# B&R Automation Studio project TD52 (part 109)

#### DefaultGTCyclic.st - Cyclic code
```iecst
(*******************************************************************************
DefaultGT		value set

This code is confidential and proprietary to the INNIO Company.
It may not be used in any form, or reproduced in any manner,
without the express written permission of the INNIO Company.
Copyright, INNIO Company, 2025

Customized modifications: -
------------------------

History:
-------
V3.99.0		18.09.2012	Denk	new
V04.03.00	02.07.2015	Denk 	Backfire device for 4 gaslines and prechamber
V04.04.00	02.12.2016	Denk 	IN_GT.tSIFA_BOV.Di added
V04.07.00   04.04.2019	Zengerer ParaFactoryDefaults in Init, against missing values at upgrade engines
V04.07.01   06.06.2019	Zengerer ParaFactoryDefaults in Init
V04.25.00	17.12.2025	Theobald With SafetyPLC the gas safety device signals will not be set

Instructions for use:
--------------------
- Default TRUE setting for not existing Di's

Outstandings:
------------

*******************************************************************************)

PROGRAM _CYCLIC

	(* Default TRUE setting for not existing Di's *)
	IN_GT.tDiffPrct_TC2.Di			:= IN_GT.tDiffPrct_TC2.Di 			OR NOT IN_GT.tDiffPrct_TC2.GoodQual;
	IN_GT.tGndFailure_TC2.Di		:= IN_GT.tGndFailure_TC2.Di 		OR NOT IN_GT.tGndFailure_TC2.GoodQual;
	IN_GT.tGT1_SafeDevOK.Di			:=(IN_GT.tGT1_SafeDevOK.Di 			OR NOT IN_GT.tGT1_SafeDevOK.GoodQual) AND NOT IN_GT.bSafetyPLC_Active; 	(* SAFETY PLC *)
	IN_GT.tGT2_SafeDevOK.Di			:=(IN_GT.tGT2_SafeDevOK.Di 			OR NOT IN_GT.tGT2_SafeDevOK.GoodQual) AND NOT IN_GT.bSafetyPLC_Active;	(* SAFETY PLC *)
	IN_GT.tFlairRdy.Di				:= IN_GT.tFlairRdy.Di 				OR NOT IN_GT.tFlairRdy.GoodQual;
	IN_GT.tRelGasPlant.Di			:= IN_GT.tRelGasPlant.Di 			OR NOT IN_GT.tRelGasPlant.GoodQual;
	IN_GT.tPr_GT_MinBefCompr.Di		:= IN_GT.tPr_GT_MinBefCompr.Di 		OR NOT IN_GT.tPr_GT_MinBefCompr.GoodQual;
	IN_GT.tT_GT_Ok.Di				:= IN_GT.tT_GT_Ok.Di 				OR NOT IN_GT.tT_GT_Ok.GoodQual;
	IN_GT.tGT_GC_Fail.Di			:= IN_GT.tGT_GC_Fail.Di 			OR NOT IN_GT.tGT_GC_Fail.GoodQual;
	IN_GT.tGT_FlairFail.Di			:= IN_GT.tGT_FlairFail.Di 			OR NOT IN_GT.tGT_FlairFail.GoodQual;
	IN_GT.tGT_FlareOpMod.Di			:= IN_GT.tGT_FlareOpMod.Di 			OR NOT IN_GT.tGT_FlareOpMod.GoodQual;
	IN_GT.tPr_PCG_Min.Di			:= IN_GT.tPr_PCG_Min.Di 			OR NOT IN_GT.tPr_PCG_Min.GoodQual;
	IN_GT.tOlShortCirc_TC2.Di		:= IN_GT.tOlShortCirc_TC2.Di 		OR NOT IN_GT.tOlShortCirc_TC2.GoodQual;
	IN_GT.tGenPrctTrip_TC2.Di		:= IN_GT.tGenPrctTrip_TC2.Di 		OR NOT IN_GT.tGenPrctTrip_TC2.GoodQual;
	IN_GT.tPr_GT1_Min.Di			:= IN_GT.tPr_GT1_Min.Di 			OR NOT IN_GT.tPr_GT1_Min.GoodQual;
	IN_GT.tPr_GT2_Min.Di			:= IN_GT.tPr_GT2_Min.Di 			OR NOT IN_GT.tPr_GT2_Min.GoodQual;
	IN_GT.tPr_GT1_Max.Di			:= IN_GT.tPr_GT1_Max.Di 			OR NOT IN_GT.tPr_GT1_Max.GoodQual;
	IN_GT.tPr_GT2_Max.Di			:= IN_GT.tPr_GT2_Max.Di 			OR NOT IN_GT.tPr_GT2_Max.GoodQual;
	IN_GT.tSafetyLoop_Eng.Di		:= IN_GT.tSafetyLoop_Eng.Di 		OR NOT IN_GT.tSafetyLoop_Eng.GoodQual;
	IN_GT.tP_GT_Max_Backfire.Di		:= IN_GT.tP_GT_Max_Backfire.Di 		OR NOT IN_GT.tP_GT_Max_Backfire.GoodQual;
	IN_GT.tPCG_GC_Fail.Di			:= IN_GT.tPCG_GC_Fail.Di 			OR NOT IN_GT.tPCG_GC_Fail.GoodQual;
	IN_GT.tPCG_GC_Oil_Min.Di		:= IN_GT.tPCG_GC_Oil_Min.Di 		OR NOT IN_GT.tPCG_GC_Oil_Min.GoodQual;
	IN_GT.tGT_BackFireDev.Di		:= IN_GT.tGT_BackFireDev.Di 		OR NOT IN_GT.tGT_BackFireDev.GoodQual;
	IN_GT.tGT1_1_BackFireDev.Di		:= IN_GT.tGT1_1_BackFireDev.Di 		OR NOT IN_GT.tGT1_1_BackFireDev.GoodQual;
	IN_GT.tGT1_2_BackFireDev.Di		:= IN_GT.tGT1_2_BackFireDev.Di 		OR NOT IN_GT.tGT1_2_BackFireDev.GoodQual;
	IN_GT.tGT1_3_BackFireDev.Di		:= IN_GT.tGT1_3_BackFireDev.Di 		OR NOT IN_GT.tGT1_3_BackFireDev.GoodQual;
	IN_GT.tGT1_4_BackFireDev.Di		:= IN_GT.tGT1_4_BackFireDev.Di 		OR NOT IN_GT.tGT1_4_BackFireDev.GoodQual;
	IN_GT.tPCbComp_BackFireDev.Di 	:= IN_GT.tPCbComp_BackFireDev.Di 	OR NOT IN_GT.tPCbComp_BackFireDev.GoodQual;
	IN_GT.tPCaComp_BackFireDev.Di	:= IN_GT.tPCaComp_BackFireDev.Di 	OR NOT IN_GT.tPCaComp_BackFireDev.GoodQual;
	IN_GT.tRelMainGVext.Di			:= IN_GT.tRelMainGVext.Di 			OR NOT IN_GT.tRelMainGVext.GoodQual;
	IN_GT.tPr_PCGBefComp_Lo.Di		:= IN_GT.tPr_PCGBefComp_Lo.Di 		OR NOT IN_GT.tPr_PCGBefComp_Lo.GoodQual;
	IN_GT.tT_PCGAfComp_Hi.Di		:= IN_GT.tT_PCGAfComp_Hi.Di 		OR NOT IN_GT.tT_PCGAfComp_Hi.GoodQual;
	IN_GT.tGT_AirSupply_LoLo.Di		:= IN_GT.tGT_AirSupply_LoLo.Di		OR NOT IN_GT.tGT_AirSupply_LoLo.GoodQual;
	IN_GT.tPr_GT1_1_Max.Di			:= IN_GT.tPr_GT1_1_Max.Di 			OR NOT IN_GT.tPr_GT1_1_Max.GoodQual;
	IN_GT.tPr_GT1_2_Max.Di			:= IN_GT.tPr_GT1_2_Max.Di 			OR NOT IN_GT.tPr_GT1_2_Max.GoodQual;
	IN_GT.tPr_GT1_3_Max.Di			:= IN_GT.tPr_GT1_3_Max.Di 			OR NOT IN_GT.tPr_GT1_3_Max.GoodQual;
	IN_GT.tPr_GT1_4_Max.Di			:= IN_GT.tPr_GT1_4_Max.Di 			OR NOT IN_GT.tPr_GT1_4_Max.GoodQual;
	IN_GT.tPr_GT1_1_Min.Di			:= IN_GT.tPr_GT1_1_Min.Di 			OR NOT IN_GT.tPr_GT1_1_Min.GoodQual;
	IN_GT.tPr_GT1_2_Min.Di			:= IN_GT.tPr_GT1_2_Min.Di 			OR NOT IN_GT.tPr_GT1_2_Min.GoodQual;
	IN_GT.tPr_GT1_3_Min.Di			:= IN_GT.tPr_GT1_3_Min.Di 			OR NOT IN_GT.tPr_GT1_3_Min.GoodQual;
	IN_GT.tPr_GT1_4_Min.Di			:= IN_GT.tPr_GT1_4_Min.Di 			OR NOT IN_GT.tPr_GT1_4_Min.GoodQual;
	IN_GT.tSIFA_BOV.Di              := IN_GT.tSIFA_BOV.Di       		OR NOT IN_GT.tSIFA_BOV.GoodQual;

END_PROGRAM
```

#### DefaultGTInit.st - Initialization code
```iecst
(********************************************************************
 * COPYRIGHT -- INNIO Company
 ********************************************************************
 * Program: DefaultGT
 * File: DefaultGTInit.st
 * Author: 105046866
 * Created: September 18, 2012
 ********************************************************************
 * Implementation of program DefaultGT
 ********************************************************************)

PROGRAM _INIT

	(* Internal setting *)
	bTestEnabled := FALSE;

	(* V4.07 Para defaults against missing values at upgrade engines *)
	ParaFactoryDefault.iGasTrain_Type 			:= 1;
	ParaFactoryDefault.iGasTrain_Upstream_Type	:= 0;
	ParaFactoryDefault.rGasImp_Prescaling		:= 1;

END_PROGRAM
```

### Program Logical/Gastrain/gasum (IEC) - Gasumschaltung

#### gasumCyclic.st
```iecst
(***************************************************************************
gasum			GASUMSCHALTUNG/GASMISCHBETRIEB MIT KLAPPEN/VENTILEN BZW. TECJET

This code is confidential AND proprietary to the INNIO Company.
It may NOT be used in any form, OR reproduced in any manner,
without the express written permission of the INNIO Company.
Copyright, INNIO Company, 2019

Customized modifications: -
------------------------

History:
-------
V0.1	03.07.98/Pa		erstellt
        24.11.98/Pa		korrekturlesung
V170	06.04.02/LH		überarbeitet
V180	21.01.03/LH		Fehler bei Umschaltung im Stillstand ausgebessert
V183	18.09.03/LH		Kontaktplan --> strukturierten Text
 		02.10.03/LH		Gasmischbetrieb
V2071	22.11.04/LH		Schliessen der entsprechenden Gasstrecke bei Erreichen einer Endlage
                   		Blockierung Mischgasstart
		07.02.05/LH		Gasstrecke nicht mehr anwählbar wenn gestört
		03.03.05/LH		neue Variable "GASUM" eingeführt
V2071b	28.06.05/LH		Task überarbeitet
V210	18.10.04/LH		neu: Mischgasverhältnis manuell einstellbar
V220	28.03.07/LH		Task überarbeitet
V2201	08.08.07/LH		Leistung absenken vor Öffnen der 2. Gasstrecke bei TecJet
V230	16.01.08/LH		Hinweis für Leistungsabsenkung
V2311a	13.05.08/LH		Leistungsabsenkung aus Mischgas wenn Gasmischverhältnis aus Endlage geht
V2.50.0	25.03.2009 		Lettenb.	ssPowerSetpointLimit2 was ssPowerSetpointLimit1 (gasmix->res.2)
V2.50.1 08.07.2009 		Lett./LH Fehler bei Schritt30, bCrossOver und P_FUG ausgebessert
V2.60.0	06.10.2009 		Lettenb	task activation added
V2.60.1	20.01.2010 		lettenb.	INIT: M_GASV1 preset TRUE was FALSE, init vars reduced
V3.20.0	30.09.2010 		Maier(BuR)	M_GSEIN replaced with GCB_ON
V3.99	21-09-2013		Denk 	       	generated for modular software
V3.99.1	14-03-2013		Denk 	       	rFeedbFlap1,rFeedbFlap2,rGT_RatioMix_Set changed from Para to IN-structure
V4.00.00 25-02-2014		Denk/Zengerer  	new interface IN_GT.bGT_SelectRatioMix for DI 'MISCH', FA_M_GASV1, V2 parameter limitation
V4.03.00 29-05-2015		Denk	       	Bugfix, FA_M_GASV2.Hy soll immer 0 sein. Wie bei XT3.
		 02-07-2015		Denk 			Bugfix, 3321 NOT activ when gastrain 2 is active. NOT was missing --> NOT MM2VIS.bMsg1028
		 								Warnings FOR 4 gaslines bMsg2694-2696 added
V4.04.00 06.02.2017		Denk			Bugfix, IN_GT.bIdx_Leanox_Act deleted, changed to IN_GT.bLeanox_Active
V4.05.00 12-10-2017		Zengerer  		Prepare vor standard with tCustAnaIn[1] or IN_GT.rGT_RatioMix_Set, to select the customized setpoint value for ssRatioMix  [0-1]
V4.11.00 17-03-2022		Zuschnig	Use standard label from customized modul for gasmixing setpoint
		 18-03-2022		Zuschnig	Removed fixed spare parameter and customized analog input
V4.13.00 20-06-2023		Zuschnig  	Added standardized AI input for gas mixing ratio
		 20-12-2023		Zuschnig	Prevent division by zero

Instructions for use:
--------------------
activate task if used with Parameter

Outstandings:
------------

****************************************************************************)

(* Übersicht Gasumschaltung *)

(*
           +---------------------------------+                              Umschaltung mit Klappen/Ventilen
           !                                 !                              ohne Rückmeld. und guter Gasqualität
           V                                 V
    +-------------+   +-------------+   +-------------+   +-------------+   Umschaltung mit Klappen/Ventilen
    ! GAS1_2|GAS1 !<->!    GAS2     !<->!    GAS4     !<->!    GAS3     !   ohne Rückmeldung und
    +-------------+   +-------------+   +-------------+   +-------------+   schlechter Gasqualität
           A                                                      A
           !          +-------------------------------+           !         Umschaltung bzw. Gasmischbetrieb mit
           +--------->!           GAS1_3              !<----------+         Klappen/Ventilen mit Rückmeldung
                      +-------------------------------+                     oder mit TecJet

****************************************************************************)
PROGRAM _CYCLIC

(*task activation *)
IF NOT Para.bGT_MixActive THEN
	RETURN;
END_IF

	IF	NOT Para.bTJ_Exist	THEN
		T_GAS1;										(* Klappen-Umschaltzeit [sec], Parameter Eingabe in sec *)
		T_GAS2;										(* Klappen-Umschaltzeit [sec], Parameter Eingabe in sec *)
		T_GAS3;										(* Klappen-Umschaltzeit [sec], Parameter Eingabe in sec *)
		T_GAS4;										(* Klappen-Umschaltzeit [sec], Parameter Eingabe in sec *)
		T_GAS1_4;									(* Klappen-Umschaltzeit [sec], Parameter Eingabe in sec *)
		T_GAS4_1;									(* Klappen-Umschaltzeit [sec], Parameter Eingabe in sec *)
		T_IMPULS;									(* Stellimpuls Klappen  [sec], Parameter Eingabe in sec *)
		T_PAUSE;									(* Pausenzeit Klappen   [sec], Parameter Eingabe in sec *)

		FA_GAS1_2.In		:=	X_GMISCH_2;			(* Gas quality [0-1 = 0-100%] *)
		FA_GAS1_2.Gw		:=	0;					(* GW hohe Qual. [0-1 = 0-100%], Parameter Eingabe in 0-100% *)
		FA_GAS1_2.Hy		:=	0;					(* HY hohe Qual. [0-1 = 0-100%], Parameter Eingabe in 0-100% *)
		FA_GAS1_2;
		GAS1_2_HQ			:=	FA_GAS1_2.Q;		(* GAS1_2 mit hoher Qualität *)

		mit_RM				:=	FALSE;				(* Rückmeldung von Klappen/Ventilen vorhanden *)
		RM_KL1				:=	0;					(* RM Klappe/Ventil Gasstrecke 1 *)
		RM_KL2				:=	0;					(* RM Klappe/Ventil Gasstrecke 2 *)

	END_IF;
	(* bis hier eventuell löschen ------------------------------------------------------------------------------------------------------- *)

	(* Gas mixing setpoint from MM Customized, or directliy connected here with Customized AI[x]  *)
	IF  IN_GT.bOptGT_RatioMix_Set THEN
		X_SOLLW			:=	REAL_TO_INT(LIMIT(0.0, IN_GT.rGT_RatioMix_Set, 1.0) * 1000);	(* Ratio mix from customized module -> 0 - 1 = 0 - 100% *)
	ELSE
		X_SOLLW			:=	REAL_TO_INT(LIMIT(0.0, IN_GT.tGT_RatioMix_Set.Ai, 1.0) * 1000); (* Ratio mix from AI standard label -> 0 - 1 = 0 - 100% *)
	END_IF

	MISCH				:=  IN_GT.tGT_SelectRatioMix.Di;									(* Digital input to select gas mixing (1-3 or 1_2-3) *)
	GUMSCH 				:= 	IN_GT.tGT_TypSwitch.Di;											(* Digital input to select gas type switching *)

	FA_M_GASV1.In		:=	REAL_TO_INT(OUT_GT.rGT_RatioMix * 1000);						(* MAX-Grenzwert Mischrate *)
	FA_M_GASV1.Gw		:=	1000;															(* GW Mischrate [0-1000 = 100%], Parameter Eingabe in 0-100% *)
	FA_M_GASV1.Hy		:=	5;																(* HY Mischrate [0-1000 = 100%], Parameter Eingabe in 0-100% *)
	FA_M_GASV1;																				(* --> Schliessen Gasventil 1 *)

	FA_M_GASV2.In		:=	REAL_TO_INT(OUT_GT.rGT_RatioMix * 1000);						(* MIN-Grenzwert Mischrate *)
	FA_M_GASV2.Gw		:=	0;																(* GW Mischrate [0-1000 = 100%], Parameter Eingabe in 0-100% *)
	FA_M_GASV2.Hy		:=	5;																(* HY Mischrate [0-1000 = 100%], Parameter Eingabe in 0-100% *)
	FA_M_GASV2;																				(* --> Schliessen Gasventil 2 *)

	(* Copy of input variables to local *)			//!!! new
	ssRatioMix 			:= REAL_TO_INT(OUT_GT.rGT_RatioMix * 1000);
	M_BTRB 				:= IN_GT.tEng_Run.Do;
	GCB_ON 				:= IN_GT.tGCB_On.Di;
	M_GASV 				:= OUT_GT.bGV_On;
	AUTGAS				:= OUT_GT.bSelGasTypAut;
	GAS1_2_MAN			:= OUT_GT.bSelGasTyp0;
	GAS1_3_MAN			:= OUT_GT.bSelGasTypMix;
	GAS1				:= OUT_GT.bSelGasTyp1;
	GAS2				:= OUT_GT.bSelGasTyp2;
	GAS3				:= OUT_GT.bSelGasTyp3;
	GAS4				:= OUT_GT.bSelGasTyp4;
	bLeanoxActive		:= IN_GT.bLeanox_Active;
	l_einst_a			:= IN_GT.bLeanox_Man;
	M_NANF				:= IN_GT.bEng_Dem_EPS;
	M_GDMI1W			:= MM2VIS.bMsg3221;
	M_GDMI1_1W			:= MM2VIS.bMsg2694;
	M_GDMI1_2W			:= MM2VIS.bMsg2695;
	M_GDMI1_3W			:= MM2VIS.bMsg2696;
	M_GDMI2W			:= MM2VIS.bMsg3222;
	anz_gasart			:= INT_TO_USINT(Para.iIdx_Gastyp);
	bTecJetOn			:= Para.bTJ_Exist;
	GASV1				:= OUT_GT.tGV1_Open.Do;
	GASV2				:= OUT_GT.tGV2_Open.Do;
	p_ist				:= REAL_TO_INT(IN_GT.rP_Act_Norm_Filt * IN_GT.rP_Nom);
	bSetMix_Man			:= bGT_RatioMix_Man_Set;						// From Visu
	bMisch1_2_Man		:= bGT_QualMix_Man_Set;							// From Visu
	ssSetMix_Man		:= REAL_TO_INT((rGT_RatioMix_Man_Set) * 1000);	// From Visu
	KL1_AUF				:= IN_GT.tGT_Flap1_Opened.Di;					//will be no IN in future
	KL1_ZU				:= IN_GT.tGT_Flap1_Closed.Di;					//will be no IN in future
	KL2_AUF				:= IN_GT.tGT_Flap2_Opened.Di;					//will be no IN in future
	KL2_ZU				:= IN_GT.tGT_Flap2_Closed.Di;					//will be no IN in future
	GAS1_2				:= OUT_GT.bGT_Ipol12Active;

	//There will be NO spare power reduction in future. One standard for gasmixing
	//--> required setpoint will be setted via OUT_GT.rP_Red_GasSwitch in %
	sel_PowerSetpointLimit := 1;												    				(*Auswahl Reserve-Red: 1 = P-Red Reserve 1
																										 					2 = P-Red Reserve 2
																															3 = P-Red Reserve 3 *)
	ssPowerSetpointLimit:=  4000; 																	(* Text: P_401 !     *)(* Reduktionsleistung für Öffnen 2. Gasstr.[kW] *)
																									(* P_40 Text2! *)

//	TOF_FUGITIV.PT 		:= 	INT_TO_UDINT(LIMIT(5, SPS_REZP1, 5))*100;								//existing code
	TOF_FUGITIV.PT 		:= 	500;	    															(* Verweilzeit auf Reduktionleistung [sec], Parameter Eingabe in sec *)
	TON_P_FUG.PT		:=	200;																	(* Beruhigungzeit bei Erreichen von Pred [0,01sec] *)

	T_TJ				:=	10;																		(* Änderungsgeschwindigkeit Mischrate [promill/sec] *)

	GU_TJ				:=	bTecJetOn;																(* Gasumschaltung mit TecJet *)
	GASUM				:=	TRUE;																	(* Freigabe Gasumschaltung *)
	GAS1_3				:=	GU_TJ OR mit_RM;														(* Freigabe Gasmischung *)
	bGasMixture			:=	GU_TJ AND GASUM;														(* Freigabe Mischgas für VISU (Vers. > 2.10 --> "engine data") *)

						(* Auswahl Treibgasart *)

	FG_MIX				:=	M_BTRB AND (GCB_ON OR FG_MIX);						(* Freigabe Mischgasbetrieb *)

	IF	NOT FG_MIX	THEN
						MISCH				:=	0;
						IF	M_GASV	THEN										(* Gasart fixieren! *)
											GUMSCH				:=	GUMSCH_OLD;
						ELSE				GUMSCH_OLD			:=	GUMSCH;
						END_IF;
	END_IF;

	MISCHGAS			:=	(AUTGAS AND     MISCH OR GAS1_3_MAN)AND(GAS1_3 OR   bLeanoxActive) AND NOT l_einst_a AND NOT M_NANF AND FG_MIX ;

	GASSTR_1			:=	(AUTGAS AND NOT MISCH AND NOT GUMSCH OR(GAS1       AND NOT GAS1_2)
	                                                             OR(GAS1_2_MAN AND     GAS1_2))AND NOT l_einst_a AND NOT M_NANF;
	GASSTR_2			:=	(AUTGAS AND NOT MISCH AND     GUMSCH OR GAS3                      )AND NOT l_einst_a      OR M_NANF;

	IF	(M_GDMI1W OR M_GDMI1_1W OR M_GDMI1_2W OR M_GDMI1_3W) AND ANW_GST2	THEN	(* Gasstrecke 1 nicht anwählbar! *)
						MISCHGAS			:=	0;
						GASSTR_1			:=	0;
						GASSTR_2			:=	1;
	END_IF;

	IF	M_GDMI2W AND NOT UW_GST2 OR NOT(anz_gasart > 2)	THEN						(* Gasstrecke 2 nicht anwählbar! *)
						MISCHGAS			:=	0;
						GASSTR_1			:=	1;
						GASSTR_2			:=	0;
	END_IF;

						(* Schrittkette *)

	CASE	step OF	00:	(* Initialisierung (GUI_0) *)
						IF	 ssRatioMix = 0 AND bTecJetOn OR KL1_AUF AND KL2_AUF	THEN
											step				:=	10;			(* 10 = GAS1 / 20 = GAS3 *)
	(* bis hier bearbeiten -------------------------------------------------------------------------------------------------------------- *)
											IF	bTecJetOn	THEN
																step				:=	10;
											END_IF;
											GUI_7				:=	1;			(* Initialisierung abgeschlossen ! *)
						END_IF;

					10:	(* Treibgas 1 (GU2_7) *)
						IF	 (GASSTR_2 OR MISCHGAS) AND GAS1_3	THEN
											step				:=	11;
						ELSIF GASSTR_2 AND NOT GAS1_3	THEN
											step				:=	12;
						END_IF;
						IF	  GASSTR_2 AND M_NANF AND NOT GCB_ON AND KL2_AUF AND NOT GU_TJ	THEN
											step				:=	20;
						END_IF;

					11:	(* Treibgas 1 --> Mischgas (GU13_0) *)
						IF	(KL2_ZU AND NOT GU_TJ) OR NOT M_GASV OR P_FUG	THEN
											step				:=	30;
						END_IF;

					12:	(* Schliessen Klappe 2 (GU1_0) *)
						IF	KL2_ZU OR NOT M_GASV	THEN
											step				:=	13;
						END_IF;

					13:	(* Gasart 1 (GU1_1) *)
						IF	(T_GAS1_OK AND NOT GAS1_2_HQ) OR NOT M_GASV	THEN
											step				:=	14;
						END_IF;
						IF	(T_GAS1_4_OK AND GAS1_2_HQ) OR KL2_AUF	THEN
											step				:=	15;
						END_IF;

					14:	(* Gasart 2 (GU1_2) *)
						IF	KL2_AUF OR (T_GAS1_4_OK AND GAS1_2_HQ)	THEN
											step				:=	15;
						ELSIF NOT T_GAS1_4_OK AND GAS1_2_HQ	THEN
											step				:=	13;
						END_IF;

					15:	(* Gasart 4 (GU1_3) *)
						IF	T_GAS4_OK OR NOT M_GASV	THEN
											step				:=	16;
						ELSIF NOT KL2_AUF AND NOT GAS1_2_HQ	THEN
											step				:=	14;
						END_IF;

					16:	(* Gasart 3 (GU1_4) *)
						IF	KL1_ZU OR NOT M_GASV	THEN
											step				:=	20;
						END_IF;

					17:	(* Öffnen Klappe 2 (GU31_0) *)
						IF	KL2_AUF OR GU_TJ	THEN
											step				:=	18;
						END_IF;

					18:	(* Schliessen Klappe 1 (GU31_1) *)
						IF	KL1_ZU OR NOT M_GASV OR GU_TJ	THEN
											step				:=	19;
						END_IF;

					19:	(* Mischgas --> Treibgas 2 (GU31_2) *)
						IF	ssRatioMix = 1000 OR NOT GU_TJ	THEN
											step				:=	20;
						ELSIF	MISCHGAS OR GASSTR_1	THEN
											step				:=	30;
						END_IF;

					20:	(* Treibgas 2 (GU1_7) *)
						IF	 (MISCHGAS OR GASSTR_1) AND GAS1_3	THEN
											step				:=	21;
						ELSIF GASSTR_1 AND NOT GAS1_3	THEN
											step				:=	22;
						END_IF;

					21:	(* Treibgas 2 --> Mischgas (GU23_0) *)
						IF	KL1_ZU AND NOT GU_TJ OR NOT M_GASV OR P_FUG	THEN
											step				:=	30;
						END_IF;

					22:	(* Schliessen Klappe 1 (GU2_0) *)
						IF	KL1_ZU OR NOT M_GASV	THEN
											step				:=	23;
						END_IF;

					23:	(* Gasart 3 (GU2_1) *)
						IF	T_GAS3_OK OR NOT M_GASV OR KL1_AUF	THEN
											step				:=	24;
						END_IF;

					24:	(* Gasart 4 (GU2_2) *)
						IF	KL1_AUF	THEN
											IF	NOT GAS1_2_HQ	THEN
																step				:=	25;
											ELSIF	T_GAS4_1_OK OR NOT M_GASV	THEN
																step				:=	26;
											END_IF;
						END_IF;

					25:	(* Gasart 2 (GU2_3) *)
						IF	T_GAS2_OK OR (T_GAS4_1_OK AND GAS1_2_HQ) OR NOT M_GASV	THEN
											step				:=	26;
						ELSIF NOT T_GAS4_1_OK AND GAS1_2_HQ	THEN
											step				:=	24;
						END_IF;

					26:	(* Gasart 1 (GU2_4) *)
						IF	KL2_ZU OR NOT M_GASV	THEN
											step				:=	10;
						ELSIF NOT T_GAS2_OK AND NOT GAS1_2_HQ	THEN
											step				:=	25;
						END_IF;

					27:	(* Öffnen Klappe 1 (GU32_0) *)
						IF	KL1_AUF OR GU_TJ	THEN
											step				:=	28;
						END_IF;

					28:	(* Schliessen Klappe 2 (GU32_1) *)
						IF	KL2_ZU OR NOT M_GASV OR GU_TJ	THEN
											step				:=	29;
						END_IF;

					29:	(* Mischgas --> Treibgas 1 (GU32_2) *)
						IF	ssRatioMix = 0 OR NOT GU_TJ	THEN
											step				:=	10;
						ELSIF	GASSTR_2 OR MISCHGAS	THEN
											step				:=	30;
						END_IF;

					30:	(* Mischgas (GU3_7) *)
						IF		GASSTR_2	THEN
											step				:=	17;
						ELSIF	GASSTR_1	THEN
											step				:=	27;
						END_IF;
						IF	(X_SOLLW > (FA_M_GASV2.Gw + FA_M_GASV2.Hy)) AND NOT GASV2 AND M_GASV AND NOT P_FUG AND GU_TJ	THEN
											step				:=	11;
						END_IF;
						IF	(X_SOLLW < (FA_M_GASV1.Gw - FA_M_GASV1.Hy)) AND NOT GASV1 AND M_GASV AND NOT P_FUG AND GU_TJ	THEN
											step				:=	21;
						END_IF;

	END_CASE;

						(* Schrittkettenmerker *)

	zw					:= 1;
	FOR	i				:= 1 TO step	BY 1 DO
						zw				:=	zw * 2;
	END_FOR;
	FA_CONV_1.Word		:= UDINT_TO_UINT(zw);
	FA_CONV_1;

	zw					:= 1;
	FOR i				:= 17 TO step	BY 1 DO
						zw				:=	zw * 2;
	END_FOR;
	IF	step < 16 THEN	zw				:=	0;
	END_IF;
	FA_CONV_2.Word		:= UDINT_TO_UINT(zw);
	FA_CONV_2;

	GUI_0				:= FA_CONV_1.Bit00;										(* Initialisierung *)
	GUI_1				:= FA_CONV_1.Bit01;										(* Initialisierung *)
	GUI_2				:= FA_CONV_1.Bit02;										(* Initialisierung *)
	GUI_3				:= FA_CONV_1.Bit03;										(* Initialisierung *)
	GUI_4				:= FA_CONV_1.Bit04;										(* Initialisierung *)
	GUI_5				:= FA_CONV_1.Bit05;										(* Initialisierung *)
	GUI_6				:= FA_CONV_1.Bit06;										(* Initialisierung *)
	muell				:= FA_CONV_1.Bit07;
	muell				:= FA_CONV_1.Bit08;
	muell				:= FA_CONV_1.Bit09;
	GU2_7				:= FA_CONV_1.Bit10;										(* Treibgas 1 *)
	GU13_0				:= FA_CONV_1.Bit11;										(* Treibgas 1 --> Mischgas *)
	GU1_0				:= FA_CONV_1.Bit12;										(* Schliessen Klappe/Ventil 2 *)
	GU1_1				:= FA_CONV_1.Bit13;										(* Gasart 1 / Gasart 1_2 *)
	GU1_2				:= FA_CONV_1.Bit14;										(* Gasart 2 *)
	GU1_3				:= FA_CONV_1.Bit15;										(* Gasart 4 *)
	GU1_4				:= FA_CONV_2.Bit00;										(* Gasart 3 *)
	GU31_0				:= FA_CONV_2.Bit01;										(* Öffnenen Klappe/Ventil 2 *)
	GU31_1				:= FA_CONV_2.Bit02;										(* Schliessen Klappe/Ventil 1 *)
	GU31_2				:= FA_CONV_2.Bit03;										(* Mischgas --> Treibgas 2 *)
	GU1_7				:= FA_CONV_2.Bit04;										(* Treibgas 2 *)
	GU23_0				:= FA_CONV_2.Bit05;										(* Treibgas 2 --> Mischgas *)
	GU2_0				:= FA_CONV_2.Bit06;										(* Schliessen Klappe/Ventil 2 *)
	GU2_1				:= FA_CONV_2.Bit07;										(* Gasart 3 *)
	GU2_2				:= FA_CONV_2.Bit08;										(* Gasart 4 *)
	GU2_3				:= FA_CONV_2.Bit09;										(* Gasart 2 *)
	GU2_4				:= FA_CONV_2.Bit10;										(* Gasart 1 / Gasart 1_2 *)
	GU32_0				:= FA_CONV_2.Bit11;										(* Öffnenen Klappe/Ventil 1 *)
	GU32_1				:= FA_CONV_2.Bit12;										(* Schliessen Klappe/Ventil 2 *)
	GU32_2				:= FA_CONV_2.Bit13;										(* Mischgas --> Treibgas 1 *)
	GU3_7				:= FA_CONV_2.Bit14;										(* Mischgas *)
	muell				:= FA_CONV_2.Bit15;

						(* Setzen der Steuerbefehle *)

	FG_GST				:=	GUI_7 AND(GU2_7 OR GU1_7 OR M_BTRB OR GU3_7 AND GAS1_3);(* Freigabe Gasstrecke (pb6!) *)

	FG_MISCH			:=	GU3_7;												(* Freigabe Gasmischregler (reg_in!)*)

	V_GVD				:=	GU23_0;												(* Vorhalte Gasverdichter *)

	ANW_GST2			:=	GU1_7 OR GU23_0 OR GU2_0;							(* Anwahl Gasstrecke 2 *)
	UW_GST2				:=	NOT(GU2_7 OR GU13_0 OR GU1_0);						(* Überwachung Gasstrecke 2 *)

	M_GASV1				:=	NOT ANW_GST2 AND(									(* Anwahl Gasventil 1 *)
							GU_TJ OR NOT KL1_ZU)AND(NOT
							GU_TJ OR NOT FA_M_GASV1.Q);
	M_GASV2				:=	UW_GST2 AND(										(* Anwahl Gasventil 2 *)
							GU_TJ OR NOT KL2_ZU)AND(NOT
							GU_TJ OR NOT FA_M_GASV2.Q);

	bCrossOver			:=	GASV1 AND GASV2 AND bTecJetOn;						(* Gasmischung aktiv für TecJet's *)

	M_AWGAS1			:=	(GU1_1 OR GU2_4 OR NOT M_GASV2)AND NOT GAS1_2;		(* Anwahl Gas1 *)
	M_AWGAS1_2			:=	(GU1_1 OR GU2_4 OR NOT M_GASV2)AND     GAS1_2;		(* Anwahl Interpolation *)
	M_AWGAS1_3			:=	(GU3_7 OR GU31_2 OR GU32_2)AND bCrossOver OR(		(* Anwahl Mischgas *)
							GU31_0 OR GU31_1 OR
							GU32_0 OR GU32_1)AND NOT bTecJetOn;

	M_AWGAS1			:=	M_AWGAS1 OR M_AWGAS1_2 OR M_AWGAS1_3;				(* Anwahl Gas1 *)
	M_AWGAS2			:=	(GU1_2 OR GU2_3);									(* Anwahl Gas2 *)
	M_AWGAS3			:=	(GU1_4 OR GU2_1 OR NOT M_GASV1);					(* Anwahl Gas3 *)
	M_AWGAS4			:=	(GU1_3 OR GU2_2);									(* Anwahl Gas4 *)

	IF	M_GASV AND (GU13_0 OR GU23_0) AND NOT bCrossOver AND bTecJetOn	THEN(* Entlasten für Öffnen anderen Gasstrecke *)
						FUGITIV				:=	1;								(* Anforderung Leistungsreduktion *)
	ELSE				FUGITIV				:=	0;
	END_IF;

	TOF_FUGITIV.IN := FUGITIV;
	TOF_FUGITIV.PT := MAX(TOF_FUGITIV.PT, ((MAX((1000 - (FA_M_GASV1.Gw - FA_M_GASV1.Hy)), ((FA_M_GASV2.Gw + FA_M_GASV2.Hy) - 0))/MAX(1, T_TJ))*100));
	TOF_FUGITIV();
	sel_PowerSetpointLimit := LIMIT(0, sel_PowerSetpointLimit, 3);
	bPowerSetpointLimit    :=((p_ist > ssPowerSetpointLimit) OR bPowerSetpointLimit) AND TOF_FUGITIV.Q AND (sel_PowerSetpointLimit > 0);

	TON_P_FUG.IN := ((p_ist <= ssPowerSetpointLimit) OR TON_P_FUG.IN) AND
					((p_ist - ssPowerSetpointLimit) < ssPowerSetpointLimit/50);
	TON_P_FUG();

	IF	TON_P_FUG.Q AND FUGITIV	THEN
						P_FUG				:=	1;								(* Reduktionsleistung erreicht *)
	ELSE				P_FUG				:=	0;
	END_IF;

	IF		GASSTR_1 OR GU32_2 OR GUI_0	THEN									(* Gasmischverhältnis für GAS1 *)
						X_SOLLW				:=	0;
	ELSIF	GASSTR_2 OR GU31_2	THEN											(* Gasmischverhältnis für GAS3 *)
						X_SOLLW				:=	1000;
	ELSE				X_SOLLW				:=	MUX(BOOL_TO_SINT(bSetMix_Man),	(* Gasmischverhältnis für Mischbetrieb *)
												X_SOLLW, ssSetMix_Man);
	END_IF;

	IF	M_GASV AND (l_einst_a OR GU13_0 OR GU23_0)	THEN						(* Gasmischverhältnis fixieren! *)
						X_SOLLW				:=	X_SOLLW_OLD;
	ELSE				X_SOLLW_OLD			:=	X_SOLLW;
	END_IF;

	IF	NOT M_GASV OR (GU31_2 AND M_NANF AND NOT GCB_ON)	THEN				(* disable ramp fub *)
						RAMPE_X_SOLLW.enable := FALSE;
	ELSE				RAMPE_X_SOLLW.enable := TRUE;							(* enable ramp fub *)
						RAMPE_X_SOLLW.Rise	 := INT_TO_UINT(					(* pos. change of gas mixture 0,1%/sec *)
												LIMIT(0,T_TJ*BOOL_TO_INT(NOT l_einst_a),10));
						RAMPE_X_SOLLW.Sink	 := INT_TO_UINT(					(* neg. change of gas mixture 0,1%/sec *)
												LIMIT(0,T_TJ*BOOL_TO_INT(NOT l_einst_a),10));
	END_IF;
	RAMPE_X_SOLLW.TC_Time:= 100;												(* FUB is working in 100ms task		*)
	RAMPE_X_SOLLW.In	 := X_SOLLW;
	RAMPE_X_SOLLW();

	OUT_GT.rGT_MixSet	:= 	INT_TO_REAL(LIMIT(0, RAMPE_X_SOLLW.Out, 1000)) / 1000;	(* Sollwert für Gasmischverhältnis *)
//	ssSetMix			:=	LIMIT(0, RAMPE_X_SOLLW.Out, 1000);						(* Sollwert für Gasmischverhältnis *)		//Existing code

						(* Steuerbefehle für Klappen/Ventile *)

	KL1AUF_1			:=	GUI_0 AND NOT GU_TJ;								(* Initialisierung *)
	KL1ZU_1				:=	GUI_0 AND NOT GU_TJ AND NULL;						(* Initialisierung *)
	KL2AUF_1			:=	GUI_0 AND NOT GU_TJ;								(* Initialisierung *)
	KL2ZU_1				:=	GUI_0 AND NOT GU_TJ AND NULL;						(* Initialisierung *)

	KL1AUF_2			:=	(GU2_1 OR GU2_2 AND NOT KL1_AUF)					(* Treibgas 2 --> Treibgas 1 (getaktet) *)
							AND NOT l_einst_a;
	KL1ZU_2				:=	(GU1_3 AND KL2_AUF OR GU1_4)						(* Treibgas 1 --> Treibgas 2 (getaktet) *)
							AND NOT l_einst_a;
	KL2AUF_2			:=	(GU1_1 OR GU1_2 OR GU1_3 AND NOT KL2_AUF)			(* Treibgas 1 --> Treibgas 2 (getaktet) *)
							AND NOT l_einst_a;
	KL2ZU_2				:=	(GU2_2 AND KL1_AUF AND GAS1_2_HQ OR GU2_3 OR GU2_4)	(* Treibgas 2 --> Treibgas 1 (getaktet) *)
							AND NOT l_einst_a;

	KL1AUF_3			:=	GU32_0 AND NOT GU_TJ AND NOT l_einst_a;				(* Mischgas --> Treibgas 1 (getaktet) *)
	KL1ZU_3				:=	GU31_1 AND NOT GU_TJ AND NOT l_einst_a;				(* Mischgas --> Treibgas 2 (getaktet) *)
	KL2AUF_3			:=	GU31_0 AND NOT GU_TJ AND NOT l_einst_a;				(* Mischgas --> Treibgas 2 (getaktet) *)
	KL2ZU_3				:=	GU32_1 AND NOT GU_TJ AND NOT l_einst_a;				(* Mischgas --> Treibgas 1 (getaktet) *)

	KL1AUF_4			:=	KL1AUF_2 AND NOT M_GASV OR							(* Treibgas 2 --> Treibgas 1 (direkt) *)
							GU32_0 AND NOT M_GASV AND NOT GU_TJ;				(* Mischgas --> Treibgas 1 (direkt) *)

	KL1ZU_4				:=	KL1ZU_2 AND NOT M_GASV OR							(* Treibgas 1 --> Treibgas 2 (direkt) *)
							GU31_1 AND NOT M_GASV AND NOT GU_TJ OR				(* Mischgas --> Treibgas 2 (direkt) *)
							GU1_7 AND NOT KL1_ZU AND NOT GU_TJ OR				(* Treibgas 2 (direkt) *)
							GU23_0 AND M_GASV AND NOT GU_TJ OR					(* Treibgas 2 --> Mischgas (direkt) *)
							GU2_0;												(* Treibgas 2 --> Treibgas 1 (direkt) *)

	KL2AUF_4			:=	KL2AUF_2 AND NOT M_GASV OR							(* Treibgas 1 --> Treibgas 2 (direkt) *)
							GU31_0 AND NOT M_GASV AND NOT GU_TJ OR				(* Mischgas --> Treibgas 2 (direkt) *)
							GU2_7 AND NOT KL2_AUF AND NOT GU_TJ;				(* Treibgas 1 (direkt) *)

	KL2ZU_4				:=	GU13_0 AND M_GASV AND NOT GU_TJ OR					(* Treibgas 1 --> Mischgas (direkt) *)
							GU1_0;												(* Treibgas 1 --> Treibgas 2 (direkt) *)

	KL1AUF_5			:=	GU3_7 AND NOT l_einst_a;							(* Gasmischbetrieb (Schrittregler!) *)
	KL1ZU_5				:=	GU3_7 AND NOT l_einst_a AND KL2_AUF;				(* Gasmischbetrieb (Schrittregler!) *)
	KL2AUF_5			:=	GU3_7 AND NOT l_einst_a;							(* Gasmischbetrieb (Schrittregler!) *)
	KL2ZU_5				:=	GU3_7 AND NOT l_einst_a AND KL1_AUF;				(* Gasmischbetrieb (Schrittregler!) *)

	IF	GU2_7 OR GU1_7 OR (KL1_AUF AND KL2_AUF)	THEN
						count				:=	0;
	END_IF;
	IF		(GU1_1 OR GU1_2)	THEN
						IF	count > (MIN(T_GAS1, T_GAS1_4) * 10)	THEN		(* Zeit Gasart 1 *)
											T_GAS1_OK			:=	1;
						END_IF;
						IF	count > (MAX(T_GAS1_4, T_GAS1) * 10)	THEN		(* Zeit Gasart 1 mit hoher Qualität *)
											T_GAS1_4_OK			:=	1;
						END_IF;
						count				:=	count + BOOL_TO_INT(KL2AUF_2);
	END_IF;
	IF	GU1_3 AND KL2_AUF 	THEN
						IF	count > (T_GAS4 * 10)	THEN						(* Zeit Gasart 4 (Treibgas 1 --> Treibgas 2) *)
											T_GAS4_OK			:=	1;
						END_IF;
						count				:=	count + BOOL_TO_INT(KL1ZU_2);
	END_IF;
	IF	GU2_1	THEN
						IF	count > (T_GAS3 * 10)	THEN						(* Zeit Gasart 3 *)
											T_GAS3_OK			:=	1;
						END_IF;
						count				:=	count + BOOL_TO_INT(KL1AUF_2);
	END_IF;
	IF	GU2_2 AND KL1_AUF OR GU2_3 OR GU2_4	THEN
						IF	count > (MIN(T_GAS4_1, T_GAS2) * 10)	THEN		(* Zeit Gasart 4 (Treibgas 2 --> Treibgas 1) *)
											T_GAS4_1_OK			:=	1;
						END_IF;
						IF	count > (MAX(T_GAS2, T_GAS4_1) * 10)	THEN		(* Zeit Gasart 2 *)
											T_GAS2_OK			:=	1;
						END_IF;
						count				:=	count + BOOL_TO_INT(KL2ZU_2);
	END_IF;
	IF	GU2_7 OR GU1_7	THEN
						T_GAS1_OK			:=	0;
						T_GAS1_4_OK			:=	0;
						T_GAS4_OK			:=	0;
						T_GAS3_OK			:=	0;
						T_GAS4_1_OK			:=	0;
						T_GAS2_OK			:=	0;
	END_IF;

						(* Taktgenerierung für Stellbefehle *)

	IMPULS				:=	T_IMPULS * 10;
	PAUSE				:=	T_PAUSE * 10;
	IF	count_st > (IMPULS + PAUSE)	THEN
						count_st			:=	0;
	END_IF;
	IF	count_st > 0	THEN
						STELL				:=	1;
	END_IF;
	IF	count_st > IMPULS	THEN
						STELL				:=	0;
	END_IF;
	count_st			:=	count_st + 1;

						(* Stellbefehle Klappen/Ventile *)

	KL1AUF				:=	(((KL1AUF_2 OR KL1AUF_3) AND STELL) OR (KL1AUF_5 AND GAS2_MIN) OR KL1AUF_4 OR KL1AUF_1) AND NOT KL1_AUF;
	KL1ZU				:=	(((KL1ZU_2  OR KL1ZU_3)  AND STELL) OR (KL1ZU_5  AND GAS2_PLU) OR KL1ZU_4  OR KL1ZU_1)  AND NOT KL1_ZU;
	KL2AUF				:=	(((KL2AUF_2 OR KL2AUF_3) AND STELL) OR (KL2AUF_5 AND GAS2_PLU) OR KL2AUF_4 OR KL2AUF_1) AND NOT KL2_AUF;
	KL2ZU				:=	(((KL2ZU_2  OR KL2ZU_3)  AND STELL) OR (KL2ZU_5  AND GAS2_MIN) OR KL2ZU_4  OR KL2ZU_1)  AND NOT KL2_ZU;

						(* Ventilstellwerte (mA-Vorgabe) *)

	IF	KL1AUF	THEN	count1				:=	count1 + 1;
	END_IF;
	IF	KL1ZU	THEN	count1				:=	count1 - 1;
	END_IF;
	IF	KL2AUF	THEN	count2				:=	count2 + 1;
	END_IF;
	IF	KL2ZU	THEN	count2				:=	count2 - 1;
	END_IF;
	count1				:=	LIMIT(0, count1, 1000);
	count2				:=	LIMIT(0, count2, 1000);
	SW_KL1				:=	count1;
	SW_KL2				:=	count2;

						(* Rückmeldungen Ventilendstellungen *)

	IF	NOT mit_RM	THEN
						RM_KL1				:=	SW_KL1;
						RM_KL2				:=	SW_KL2;
						IF	RM_KL1 < 1		THEN
											KL1_ZU				:=	1;
						ELSE				KL1_ZU				:=	0;
						END_IF;
						IF	RM_KL1 > 999	THEN
											KL1_AUF				:=	1;
						ELSE				KL1_AUF				:=	0;
						END_IF;
						IF	RM_KL2 < 1		THEN
											KL2_ZU				:=	1;
						ELSE				KL2_ZU				:=	0;
						END_IF;
						IF	RM_KL2 > 999	THEN
											KL2_AUF				:=	1;
						ELSE				KL2_AUF				:=	0;
						END_IF;
	END_IF;

						(* Gasverbräuche (gmv_ber) *)

	GAS1_VB	:=	BOOL_TO_INT(GASV1) * (
							BOOL_TO_INT(NOT GU_TJ)*(RM_KL1 + 1000-RM_KL2*BOOL_TO_INT(GASV2)) +
							BOOL_TO_INT(GU_TJ)*(1000 - ssRatioMix));
	GAS2_VB	:=	BOOL_TO_INT(GASV2) * (
							BOOL_TO_INT(NOT GU_TJ)*(RM_KL2 + 1000-RM_KL1*BOOL_TO_INT(GASV1)) +
							BOOL_TO_INT(GU_TJ)*ssRatioMix);

	(* Leistungsreduktionen *)
	(* Power reduction gas switching for opening second gastrain *)
	IF (ssPowerSetpointLimit <= 0.0) OR (IN_GT.rP_Act_Norm_Filt = 0.0) OR (IN_GT.rP_Nom = 0.0) THEN			//new
		OUT_GT.rP_Red_GasSwitch := 0.0;
	ELSE
		OUT_GT.rP_Red_GasSwitch := 1 - LIMIT(0.0, (Para.rP_GT_SetLim / (IN_GT.rP_Act_Norm_Filt * IN_GT.rP_Nom)), 0.5);
	END_IF;

(* Copy local output variables to global *)
	bGT_MixingEna 				:= bGasMixture;				(* Visu *)
	OUT_GT.bGT2_Select 			:= ANW_GST2;
	OUT_GT.bGT_Rel 				:= FG_GST;
	OUT_GT.bGT_RelMixing		:= FG_MISCH;
	OUT_GT.bGasMixingActive		:= bCrossOver;
	OUT_GT.bGT_SelGas1			:= M_AWGAS1;
	OUT_GT.bGT_SelGas2			:= M_AWGAS2;
	OUT_GT.bGT_SelGas3			:= M_AWGAS3;
	OUT_GT.bGT_SelGas4			:= M_AWGAS4;
    OUT_GT.tGT_Flap1_Open.Do 	:= KL1AUF;			//will be no Out in future
	OUT_GT.tGT_Flap1_Close.Do	:= KL1ZU;			//will be no Out in future
	OUT_GT.tGT_Flap2_Open.Do	:= KL2AUF;			//will be no Out in future
	OUT_GT.tGT_Flap2_Close.Do	:= KL2ZU;			//will be no Out in future
	OUT_GT.bGT_TypSwhActive		:= GASUM;

END_PROGRAM
```

#### gasumInit.st
```iecst
PROGRAM _INIT

END_PROGRAM
```

#### gasum.var
```iecst
VAR
	anz_gasart : USINT; (* number of gas types *)
	AUTGAS : BOOL := 0; (* AUTOMATIK Gasumschaltung *)
	bLeanoxActive : BOOL; (* TRUE=leanox controller is active *)
	bMisch1_2_Man : BOOL; (* 1=gas quality manual *)
	bPowerSetpointLimit : BOOL;
	bTecJetOn : BOOL; (* TRUE=gas inject valves are active *)
	count : INT := 0;
	count_st : INT := 0;
	count1 : INT := 0; (* Klappensimulation *)
	count2 : INT := 0; (* Klappensimulation *)
	FA_CONV_1 : WDtoBIT;
	FA_CONV_2 : WDtoBIT;
	FA_GAS1_2 : GR_MAXR;
	FA_M_GASV1 : GR_MAX;
	FA_M_GASV2 : GR_MIN;
	FG_GST : BOOL := 0; (* Freigabe Gasstrecke *)
	FG_MISCH : BOOL := 0; (* Freigabe Gasmischregler *)
	FUGITIV : BOOL := 0; (* Anforderung Leistungsreduktion *)
	GAS1 : BOOL := 0; (* Gasart 1 *)
	GAS1_2 : BOOL; (*param.interpolation gas1 & 2 active from CH4(or CV)*)
	GAS1_2_MAN : BOOL := 0; (* Gasart 0 manuell *)
	GAS1_3_MAN : BOOL := 0; (* Mischgas manuell *)
	GAS2 : BOOL := 0; (* Gasart 2 *)
	GAS2_MIN : BOOL := 0; (* weniger Treibgas 2 *)
	GAS2_PLU : BOOL := 0; (* mehr Treibgas 2 *)
	GAS3 : BOOL := 0; (* Gasart 3 *)
	GAS4 : BOOL := 0; (* Gasart 4 *)
	GASSTR_1 : BOOL := 0; (* Anwahl Gasstrecke 1 *)
	GASSTR_2 : BOOL := 0; (* Anwahl Gasstrecke 2 *)
	GASV1 : BOOL := 0; (* Gasventil 1 *)
	GASV2 : BOOL := 0; (* Gasventil 2 *)
	GCB_ON : BOOL := FALSE; (*Generatorschalter EIN (TK#3 synchron)*)
	GU1_0 : BOOL := 0; (* Schrittkettenmerker *)
	GU1_1 : BOOL := 0; (* Schrittkettenmerker *)
	GU1_2 : BOOL := 0; (* Schrittkettenmerker *)
	GU1_3 : BOOL := 0; (* Schrittkettenmerker *)
	GU1_4 : BOOL := 0; (* Schrittkettenmerker *)
	GU1_7 : BOOL := 0; (* Schrittkettenmerker *)
	GU2_0 : BOOL := 0; (* Schrittkettenmerker *)
	GU2_1 : BOOL := 0; (* Schrittkettenmerker *)
	GU2_2 : BOOL := 0; (* Schrittkettenmerker *)
	GU2_3 : BOOL := 0; (* Schrittkettenmerker *)
	GU2_4 : BOOL := 0; (* Schrittkettenmerker *)
	GU2_7 : BOOL := 0; (* Schrittkettenmerker *)
	GU3_7 : BOOL := 0; (* Schrittkettenmerker *)
	GU13_0 : BOOL := 0; (* Schrittkettenmerker *)
	GU23_0 : BOOL := 0; (* Schrittkettenmerker *)
	GU31_0 : BOOL := 0; (* Schrittkettenmerker *)
	GU31_1 : BOOL := 0; (* Schrittkettenmerker *)
	GU31_2 : BOOL := 0; (* Schrittkettenmerker *)
	GU32_0 : BOOL := 0; (* Schrittkettenmerker *)
	GU32_1 : BOOL := 0; (* Schrittkettenmerker *)
	GU32_2 : BOOL := 0; (* Schrittkettenmerker *)
	GUI_0 : BOOL := 0; (* Schrittkettenmerker *)
	GUI_1 : BOOL := 0; (* Schrittkettenmerker *)
	GUI_2 : BOOL := 0; (* Schrittkettenmerker *)
	GUI_3 : BOOL := 0; (* Schrittkettenmerker *)
	GUI_4 : BOOL := 0; (* Schrittkettenmerker *)
	GUI_5 : BOOL := 0; (* Schrittkettenmerker *)
	GUI_6 : BOOL := 0; (* Schrittkettenmerker *)
	GUI_7 : BOOL := 0; (* Gasumschaltung INIT abgeschlossen *)
	GUMSCH : BOOL := 0; (* Gasumschaltung auf 2.tes Treibgas *)
	GUMSCH_OLD : BOOL;
	i : INT;
	IMPULS : INT; (* Stellimpuls *)
	KL1_AUF : BOOL := 0; (* RM Gasklappe 1 offen *)
	KL1_ZU : BOOL := 0; (* RM Gasklappe 1 geschlossen *)
	KL1AUF : BOOL := 0; (* GASKLAPPE 1 AUFFAHREN *)
	KL1AUF_1 : BOOL := 0; (* Klappensteuerbefehl *)
	KL1AUF_2 : BOOL := 0; (* Klappensteuerbefehl *)
	KL1AUF_3 : BOOL := 0; (* Klappensteuerbefehl *)
	KL1AUF_4 : BOOL := 0; (* Klappensteuerbefehl *)
	KL1AUF_5 : BOOL := 0; (* Klappensteuerbefehl *)
	KL1ZU : BOOL := 0; (* GASKLAPPE 1 ZUFAHREN *)
	KL1ZU_1 : BOOL := 0; (* Klappensteuerbefehl *)
	KL1ZU_2 : BOOL := 0; (* Klappensteuerbefehl *)
	KL1ZU_3 : BOOL := 0; (* Klappensteuerbefehl *)
	KL1ZU_4 : BOOL := 0; (* Klappensteuerbefehl *)
	KL1ZU_5 : BOOL := 0; (* Klappensteuerbefehl *)
	KL2_AUF : BOOL := 0; (* RM Gasklappe 2 offen *)
	KL2_ZU : BOOL := 0; (* RM Gasklappe 2 geschlossen *)
	KL2AUF : BOOL := 0; (* GASKLAPPE 2 AUFFAHREN *)
	KL2AUF_1 : BOOL := 0; (* Klappensteuerbefehl *)
	KL2AUF_2 : BOOL := 0; (* Klappensteuerbefehl *)
	KL2AUF_3 : BOOL := 0; (* Klappensteuerbefehl *)
	KL2AUF_4 : BOOL := 0; (* Klappensteuerbefehl *)
	KL2AUF_5 : BOOL := 0; (* Klappensteuerbefehl *)
	KL2ZU : BOOL := 0; (* GASKLAPPE 2 ZUFAHREN *)
	KL2ZU_1 : BOOL := 0; (* Klappensteuerbefehl *)
	KL2ZU_2 : BOOL := 0; (* Klappensteuerbefehl *)
	KL2ZU_3 : BOOL := 0; (* Klappensteuerbefehl *)
	KL2ZU_4 : BOOL := 0; (* Klappensteuerbefehl *)
	KL2ZU_5 : BOOL := 0; (* Klappensteuerbefehl *)
	l_einst_a : BOOL; (* TRUE=leanox controller in manual *)
	M_BTRB : BOOL := 0; (* Aggregat in BETRIEB *)
	M_GASV : BOOL := 0; (* Gasventile EIN *)
	M_GDMI1W : BOOL := 0; (*3221 Gasdruck 1 minimum *)
	M_GDMI1_1W : BOOL := 0; (*2694 Gasdruck 1 Linie 1 minimum *)
	M_GDMI1_2W : BOOL := 0; (*2695 Gasdruck 1 Linie 2 minimum *)
	M_GDMI1_3W : BOOL := 0; (*2696 Gasdruck 1 Linie 3 minimum *)
	M_GDMI2W : BOOL := 0; (*3222 Gasdruck 2 minimum *)
	M_NANF : BOOL := 0; (* Notstromanforderung *)
	MISCH : BOOL := 0; (* Mischgas *)
	MISCHGAS : BOOL := 0; (* Anwahl Mischgas *)
	mit_RM : BOOL := 0; (* mit RM Klappe/Ventil *)
	muell : BOOL := 0; (* GARBAGE BIT *)
END_VAR
VAR CONSTANT
	NULL : BOOL := 0; (* immer NULL *)
END_VAR
VAR
	P_FUG : BOOL := 0; (* Reduktionsleistung erreicht *)
	p_ist : INT; (* actual filtered power [kW] T= 1sec *)
	PAUSE : INT; (* Pausenzeit *)
	RAMPE_X_SOLLW : RAMPE;
	RM_KL1 : INT; (* RM Klappe/Ventil 1 *)
	RM_KL2 : INT; (* RM Klappe/Ventil 2 *)
	sel_PowerSetpointLimit : INT;
	ssPowerSetpointLimit : INT;
	ssRatioMix : INT; (* gas mixture rate after ramp fub *)
	ssSetMix_Man : INT;
	STELL : BOOL := 0; (* Stellimpuls *)
	step : INT := 0; (* Schrittvariable *)
	SW_KL1 : INT := 0; (* Sollwert Ventil 1 *)
	SW_KL2 : INT := 0; (* Sollwert Ventil 2 *)
	T_GAS1 : INT; (* Zeitwert *)
	T_GAS1_4 : INT; (* Zeitwert *)
	T_GAS1_4_OK : BOOL := FALSE;
	T_GAS1_OK : BOOL := FALSE;
	T_GAS2 : INT; (* Zeitwert *)
	T_GAS2_OK : BOOL := FALSE;
	T_GAS3 : INT; (* Zeitwert *)
	T_GAS3_OK : BOOL := FALSE;
	T_GAS4 : INT; (* Zeitwert *)
	T_GAS4_1 : INT; (* Zeitwert *)
	T_GAS4_1_OK : BOOL := FALSE;
	T_GAS4_OK : BOOL := FALSE;
	T_IMPULS : INT; (* Zeitwert *)
	T_PAUSE : INT; (* Zeitwert *)
	T_TJ : INT := 10; (* Rampenzeit Tecjet *)
	TOF_FUGITIV : TOF_10ms;
	TON_P_FUG : TON_10ms;
	X_SOLLW : INT; (* SOLLWERT Mischgasverhältnis *)
	X_SOLLW_OLD : INT;
	zw : UDINT;
END_VAR
```

### Program Logical/Gastrain/gas_rail (IEC) - gas rail control

#### gas_railCyclic.st
```iecst
(*******************************************************************************
gas_rail

This code is confidential and proprietary to the INNIO Company.
It may not be used in any form, or reproduced in any manner,
without the express written permission of the INNIO Company.
Copyright, INNIO Company, 2019

Customized modifications: -
------------------------

History:
-------
V04.03.00	20.01.2015  Denk 		Porting J920 for XT4
			07.04.2016  Denk		Change logic for A2240 ("...ja, lass es uns so machen, dass es eine Freigabebedingung gibt. 2240 soll nur auslösen, wenn es keine Messsignalstörung 2567 gibt..." E-mail 07.04.2016 Klaus Spyra)
V04.04.00	04.07.2016	Denk		Change logic for bAMM_T_GR_HiHi. Additional: AND OUT_GT.tGV1_Open.Do;
V04.05.00	20.03.2017	Denk		SWAT920: Several changes regarding new specification
V04.05.01	24.10.2017	Zingerle	Reduction with difference pressure minimum, implemented
V04.05.02	01.03.2018	Denk		Reduction with difference pressure minimum, Spec. change and validation changes
V04.05.03	23.03.2018	Denk		Perm2 change because of new Perm_GT2 file
V04.07.00	04.07.2018	Denk		Bugfix, Anzeige Leistungsreduktion Gasdruck min.
V04.10.00	05.08.2020	Zuschnig	Included 50ms filtered for boost pressure for differential pressure limit monitoring
V04.11.00	20.01.2022	Zuschnig	Update gas rail pressure power reduction

Instructions for use:
--------------------
*******************************************************************************)
PROGRAM _CYCLIC

	(*--------------------------------------------------------------*)
	(* RESET of alarms and warnings 								*)
	(*--------------------------------------------------------------*)
	bAMM_Pr_GR_I_MS			:= FALSE;
	bAMM_Pr_GR_II_MS		:= FALSE;
	bAMM_Pr_GR_I_LoLo		:= FALSE;
	bAMM_Pr_GR_I_HiHi		:= FALSE;
	bAMM_DPr_GR_I_LoLo		:= FALSE;
	bAMM_DPr_GR_I_HiHi		:= FALSE;
	bAMM_DPr_GR_I_Lo		:= FALSE;
	bAMM_DPr_GR_I_Hi		:= FALSE;
	bAMM_T_GR_MS			:= FALSE;
	bAMM_T_GR_LoLo			:= FALSE;
	bAMM_T_GR_HiHi			:= FALSE;
	bAMM_T_GR_Lo			:= FALSE;
	bAMM_T_GR_Hi			:= FALSE;
	bAMM_Pr_MGT_a_Filt_Min	:= FALSE;

	rP_norm_red_1				:= 1.0;
	rP_norm_red_2				:= 1.0;
	OUT_GT.rP_Red_Pr_GR_Norm	:= 1.0;

	(************************************************************************************************************************************)
	(************************              				  error monitoring		 	             	           **************************)
	(************************************************************************************************************************************)
	IF IN_GT.tPB2MM.bParaSetupOk THEN

		(*----------------------------------------------------------*)
		(* measurement signal failure 								*)
		(*----------------------------------------------------------*)
		bAMM_Pr_GR_I_MS		:= Para.bPr_GR_I_Exist 	AND NOT IN_GT.tPr_GR_I.GoodQual;		(* W2443 *)
		bAMM_Pr_GR_II_MS	:= Para.bPr_GR_II_Exist	AND NOT IN_GT.tPr_GR_II.GoodQual;		(* W2444 *)
		bAMM_Pr_GR_I_II_MS  := bAMM_Pr_GR_I_MS 		AND 	bAMM_Pr_GR_II_MS; 				(* A2309 *)
		bAMM_T_GR_MS		:= Para.bT_GR_Exist 	AND NOT IN_GT.tT_GR.GoodQual;			(* W2567 *)

		(* Release monitoring	*)
		xTOF_AMM_Pr_GR_I_MS(IN 	:= bAMM_Pr_GR_I_MS,	 PT:= T#10s);	(* TOF because of filtered signals *)
		xTOF_AMM_Pr_GR_II_MS(IN	:= bAMM_Pr_GR_II_MS, PT:= T#10s);
		xTOF_AMM_T_GR_MS(IN  	:= bAMM_T_GR_MS, 	 PT:= T#10s);

		bRelMon_Pr_GR_I		:= Para.bPr_GR_I_Exist 	AND NOT xTOF_AMM_Pr_GR_I_MS.Q;
		bRelMon_Pr_GR_II	:= Para.bPr_GR_II_Exist AND NOT xTOF_AMM_Pr_GR_II_MS.Q;
		bRelMon_Pr_GR_Avg	:= bRelMon_Pr_GR_I 		OR 		bRelMon_Pr_GR_II;
		bRelMon_T_GR		:= Para.bT_GR_Exist 	AND NOT xTOF_AMM_T_GR_MS.Q;

		(*----------------------------------------------------------*)
		(* check gas rail pressure sensor deviation					*)
		(*----------------------------------------------------------*)
		LCRMAF_PGR_Deviation.x := ABS(IN_GT.tPr_GR_I.Ai - IN_GT.tPr_GR_II.Ai);

		LCRMAF_PGR_Deviation();

		xGR_MAX_Deviation.In := LCRMAF_PGR_Deviation.y;
		xGR_MAX_Deviation.Gw := 0.130;	(* 130mbar *)
		xGR_MAX_Deviation.Hy := 0.03; 	(* 30mbar *)
		xGR_MAX_Deviation();

		bDevP_GR_TooHigh := xGR_MAX_Deviation.Q AND bRelMon_Pr_GR_I AND bRelMon_Pr_GR_II;

		(*----------------------------------------------------------*)
		(* gas rail pressure limit monitoring						*)
		(*----------------------------------------------------------*)
		xGR_MAX_AGRPR(In := IN_GT.tPr_GR_I.Ai, Gw := Para.rPr_GR_HiHi, Hy := 0.0);

		bAMM_Pr_GR_I_HiHi 	:= xGR_MAX_AGRPR.Q AND bRelMon_Pr_GR_I;		(* A2244 *)

		(*----------------------------------------------------------*)
		(* differential pressure limit monitoring					*)
		(*----------------------------------------------------------*)
		xGR_MAX_APDPR(In := (rPr_GR_Avg - xFILTER_R_P2s_50ms.Out), Gw := Para.rPr_GR_Diff_HiHi, Hy := 0.0);
		xGR_MIN_APDPR(In := (rPr_GR_Avg - xFILTER_R_P2s_50ms.Out), Gw := Para.rPr_GR_Diff_LoLo, Hy := 0.0);

		bAMM_DPr_GR_I_HiHi	:= xGR_MAX_APDPR.Q AND OUT_GT.tGV1_Open.Do;	(* A2248 *)
		bAMM_DPr_GR_I_LoLo	:= xGR_MIN_APDPR.Q AND IN_GT.tGCB_On.Di ;	(* A2249 *)

		(*----------------------------------------------------------*)
		(* gas rail temperature limit monitoring					*)
		(*----------------------------------------------------------*)
		xGR_MAX_WGRTP(In := IN_GT.tT_GR.Ai, Gw := (Para.rT_GR_HiHi - 5.0), Hy := 0.0);
		xGR_MIN_WGRTP(In := IN_GT.tT_GR.Ai, Gw := (Para.rT_GR_LoLo), Hy := 0.0);

		bAMM_T_GR_Hi	:= xGR_MAX_WGRTP.Q AND bRelMon_T_GR AND OUT_GT.tGV1_Open.Do;			(* W2568 *)
		bAMM_T_GR_Lo	:= xGR_MIN_WGRTP.Q AND bRelMon_T_GR AND OUT_GT.tGV1_Open.Do;			(* W2569 *)

		xGR_MAX_AGRTP(In := IN_GT.tT_GR.Ai, Gw := Para.rT_GR_HiHi, Hy := 0.0);

		bAMM_T_GR_HiHi	:= xGR_MAX_AGRTP.Q AND bRelMon_T_GR AND OUT_GT.tGV1_Open.Do;			(* A2240 *)

		(*----------------------------------------------------------*)
		(* gas rail pressure average filtered						*)
		(*----------------------------------------------------------*)
		IF 	  (NOT bRelMon_Pr_GR_I AND NOT bRelMon_Pr_GR_II) THEN	rPr_GR_Avg :=  0;
		ELSIF (NOT bRelMon_Pr_GR_I AND 	   bRelMon_Pr_GR_II) THEN	rPr_GR_Avg :=  IN_GT.tPr_GR_II.Ai;
		ELSIF (	   bRelMon_Pr_GR_I AND NOT bRelMon_Pr_GR_II) THEN	rPr_GR_Avg :=  IN_GT.tPr_GR_I.Ai;
		ELSE
			IF NOT bDevP_GR_TooHigh  THEN
				rPr_GR_Avg := (IN_GT.tPr_GR_I.Ai + IN_GT.tPr_GR_II.Ai ) / 2;
			ELSE
				IF  ABS(IN_GT.tPr_GR_I.Ai - (rPr_MGT_sp + IN_GT.rPr_Baro_Internal)) <  ABS(IN_GT.tPr_GR_II.Ai - (rPr_MGT_sp + IN_GT.rPr_Baro_Internal))  THEN
			 		rPr_GR_Avg := IN_GT.tPr_GR_I.Ai;
				ELSE
					rPr_GR_Avg := IN_GT.tPr_GR_II.Ai;
				END_IF;
			END_IF;
		END_IF;
		OUT_GT.rPr_GR_filt := rPr_GR_Avg;

		(*----------------------------------------------------------*)
		(* gas rail pressure average unfiltered						*)
		(*----------------------------------------------------------*)
		IF 	  (NOT bRelMon_Pr_GR_I AND NOT bRelMon_Pr_GR_II) THEN	rPr_GR_Avg_UF :=  0;
		ELSIF (NOT bRelMon_Pr_GR_I AND 	   bRelMon_Pr_GR_II) THEN	rPr_GR_Avg_UF :=  IN_GT.tPr_GR_II.Unfilt;
		ELSIF (	   bRelMon_Pr_GR_I AND NOT bRelMon_Pr_GR_II) THEN	rPr_GR_Avg_UF :=  IN_GT.tPr_GR_I.Unfilt;
		ELSE
			IF NOT bDevP_GR_TooHigh  THEN
				rPr_GR_Avg_UF := (IN_GT.tPr_GR_I.Unfilt + IN_GT.tPr_GR_II.Unfilt ) / 2;
			ELSE
				IF  ABS(IN_GT.tPr_GR_I.Ai- (rPr_MGT_sp + IN_GT.rPr_Baro_Internal)) <  ABS(IN_GT.tPr_GR_II.Ai - (rPr_MGT_sp + IN_GT.rPr_Baro_Internal))  THEN
			 		rPr_GR_Avg_UF := IN_GT.tPr_GR_I.Unfilt;
				ELSE
					rPr_GR_Avg_UF := IN_GT.tPr_GR_II.Unfilt;
				END_IF;
			END_IF;
		END_IF;
		OUT_GT.rPr_GR_UF := rPr_GR_Avg_UF;

		(*----------------------------------------------------------*)
		(* calculate differential pressure 							*)
		(*----------------------------------------------------------*)
		rPr_MGT_Diff := OUT_GT.rPr_GR_filt - IN_GT.rPr_Ch_P2s_Avg;

		(*------------------------------------------------------------------*)
		(* differential pressure minimum / power reduction					*)
		(*------------------------------------------------------------------*)

		(* charge pressure depending limit calculation *)
		IF bRelMon_Pr_GR_Avg AND OUT_GT.tGV1_Open.Do THEN
			xGR_MIN_Red1_DP(In := (rPr_MGT_Diff / xSigScal_R_DPr_MGT_sp.Y_SCAL), Gw := Perm2.rDPr_limit_pgr_Pred, Hy := rHy_GR_MIN);
			IF xGR_MIN_Red1_DP.Q THEN
				OUT_GT.rP2s_red_1 := (OUT_GT.rPr_GR_filt - (Perm2.rDPr_limit_pgr_Pred * xSigScal_R_DPr_MGT_sp.Y_SCAL));
				rP_norm_red_1	  := LIMIT(0.0, (IN_GT.rP_el_max_red / MAX(1, IN_GT.rP_Nom)), 1.0);
			ELSE
				rP_norm_red_1 := 1.00;
			END_IF;

			IF Para.bPr_GR_red_Exist THEN
				IF ((Para.rPr_GR_red_start - IN_GT.tPr_MGT_a_Filt.Ai) * Para.rP_Pr_GR_red_rate) < 1.0 THEN
					rP_norm_red_2 := LIMIT(0.0, (1 - ((Para.rPr_GR_red_start - IN_GT.tPr_MGT_a_Filt.Ai) * Para.rP_Pr_GR_red_rate)), 1.0);
				ELSE
					rP_norm_red_2 := 1.00;
				END_IF;
			ELSE
				rP_norm_red_2 := 1.00;
			END_IF;

			IF IN_GT.tGCB_On.Di THEN
				OUT_GT.rP_Red_Pr_GR_Norm :=	MIN(rP_norm_red_1, rP_norm_red_2);
			ELSE
				OUT_GT.rP_Red_Pr_GR_Norm	:= 1.0;
			END_IF;

			IF ((IN_GT.tPr_MGT_a_Filt.Ai - (rPr_GR_Avg - IN_GT.rPr_Baro_Internal)) < rPr_GR_Threshold) THEN
				xTP_Pr_MGT_a_Filt_Min(IN := TRUE, PT := T#2s);
			ELSE
				xTP_Pr_MGT_a_Filt_Min(IN := FALSE, PT := T#2s);
			END_IF;

			bAMM_Pr_MGT_a_Filt_Min := xTP_Pr_MGT_a_Filt_Min.Q;
		ELSE
			xTP_Pr_MGT_a_Filt_Min(IN := FALSE, PT := T#2s);
		END_IF;

	END_IF;

END_PROGRAM
```

#### gas_railInit.st
```iecst
(*******************************************************************************
gas_rail		gas rail  					(INIT)

This code is confidential AND proprietary to the INNIO Company.
It may NOT be used in any form, or reproduced in any manner,
without the express written permission of the INNIO Company.
Copyright, INNIO Company, 2019

Customized modifications: -
------------------------

History:
-------
V04.03.00.00  20.01.2015  Denk 		Porting J920 FOR XT4
V04.12.00.00  23.08.2022  Zuschnig	Initialize standard value for power redcution gas rail pressure

Instructions FOR use:
--------------------
*******************************************************************************)
PROGRAM _INIT

	(* check gas pressure sensor deviation *)
	LCRMAF_PGR_Deviation.enable	:= TRUE;	(* *)
	LCRMAF_PGR_Deviation.base	:= 5;		(* *)

	(* Initialize standard value fr power redcution gas rail pressure *)
	IF Perm2.rDPr_limit_pgr_Pred = 0 THEN	Perm2.rDPr_limit_pgr_Pred := 0.7;	END_IF;

END_PROGRAM
```

#### gas_rail.var
```iecst
VAR
	bRelMon_Pr_GR_I : BOOL := FALSE; (*Release monitoring gas sensor 1*)
	bRelMon_Pr_GR_II : BOOL := FALSE; (*Release monitoring gas sensor 2*)
	bRelMon_T_GR : BOOL := FALSE; (*Release monitoring gas rail temperature*)
	LCRMAF_PGR_Deviation : LCRMovAvgFlt;
	xGR_MAX_AGRPR : GR_MAXR := (0); (*FuB*)
	xGR_MAX_AGRTP : GR_MAXR := (0); (*FuB*)
	xGR_MAX_APDPR : GR_MAXR := (0); (*FuB*)
	xGR_MAX_WGRTP : GR_MAXR := (0); (*FuB*)
	xGR_MIN_APDPR : GR_MINR := (0); (*FuB*)
	xGR_MIN_WGRTP : GR_MINR := (0); (*FuB*)
	xTOF_AMM_Pr_GR_II_MS : TOF := (0); (*FuB*)
	xTOF_AMM_Pr_GR_I_MS : TOF := (0); (*FuB*)
	xTOF_AMM_T_GR_MS : TOF := (0); (*FuB*)
	xGR_MAX_Deviation : GR_MAXR;
	rP_norm_red_1 : REAL; (*power reduction boost pressure of the limited power of nominal power  *)
	rP_norm_red_2 : REAL; (*power reduction derating curve for the engine of nominal power  *)
	xGR_MIN_Red1_DP : GR_MINR; (* GR_MIN for power reduction GR *)
	rHy_GR_MIN : REAL := 0.25; (* Gas train diff pressure for power reduction hysteresis *)
	rPr_GR_Threshold : REAL := 0.05; (* Threshold for difference between main gas pressure after filter and gas rail pressure [bar] *)
	xTP_Pr_MGT_a_Filt_Min : TP; (* TP for difference between main gas pressure after filter and gas rail pressure minimum *)
END_VAR
```

### Program Logical/Gastrain/gas_train (IEC) - gas train control

#### gas_trainCyclic.st
```iecst
(*******************************************************************************
gas_train

This code is confidential and proprietary to the INNIO Company.
It may not be used in any form, or reproduced in any manner,
without the express written permission of the INNIO Company.
Copyright, INNIO Company, 2019

Customized modifications: -
------------------------

History:
-------
V3.30.0		06.11.2014  Tinello	NEW specification
V4.03.00  	13.11.2014  Mari 		Porting J920 FOR XT4
			09.02.2014  Denk 		Bugfix, monitoring OF load rejection
			02.06.2015  Denk		MM2VIS.rPr_PCGT_sp, MM2VIS.rPr_MGT_sp now in gas_train task
V4.04.00	03.07.2016	Denk		Blow off valve Open, Spec. change: gasrail pressure > baro pressure + 80mbar (IN_GT.rPr_Baro_Internal + 0.08)
			04.08.2016	Denk		Bugfix, Filterung charge pressure
			15.09.2016	Denk 		set/actual gas pressure comparison, hard coded values changed
			20.10.2016	Tinello		A2271 deleted / A2261 change limit from 60mbar to 100mbar
V4.05.00	24.04.2017	Denk		SWAT 920 Rel.2, A2247 deleted, W2462 new, B2927 new, OUT_GT.bAMM_Pr_MGT_a_Filt_BlockStart new
									SWAT 920 Rel.2, A3377 active > 2MW
			10.07.2017	Denk		SWAT 920 Rel.3, A2257 deleted, W2465 new, B2928 new, OUT_GT.bAMM_Pr_PCGT_a_Filt_BlockStart new
V4.07.00	30.04.2018	Denk		SWAT 920 Rel.5, change A2289 to W2570
									SWAT 920 Rel.5,	deactivation of A3376 when pressure based control is active
									SWAT 920 Rel.5,	W3445 delay time
V4.07.00	10.12.2018	Zengerer 	Gas valve position detection for Requisition standardisation
V4.07.01	28.08.2019	Zengerer 	Upstream Gas valve tGV_Upstream_Open
V4.09.00BETA 02.10./10.07.2019	Ze 	iGasTrain_Upstream_Type.0 corr. basisupdate
		 	21.08.2019	Zengerer 	Alternative path, if NO selection bit from Para.iGasTrain_Upstream_Type is active
		 	19.11.2019	Zengerer 	Customer Main Gas Valve control and position feedback according to updated spec from Lang Thomas
V4.10.00    05.08.2020  Zuschnig    Added control of dome blow off valve
			07.12.2020	Zengerer	IN_GT.tFastStartReq for change according to issue #
V4.11.00	22.06.2021	Arnold		data center serialization: calculation of rPr_MGT_sp based on IN_GT.rPr_Leanox_Set; DBOV different hysteresis and time delay
			20.01.2022	Zuschnig	Update A2289 - Compressed air supply failure
			11.02.2022 	Zuschnig	Remove engine demand for release of upstream gas valve
V4.12.00	22.01.2023	Zuschnig	Add H2 content processing and detection of measurement failure
V4.14.00	06.11.2024	Kafka		fast gastrain for Gen2 type9

Instructions for use:
--------------------
Use UPSTREAM MAIN GAS VALVE OPTION 0 or 1 only (OUT_GT.tGV_Upstream_Open)
UPSTREAM MAIN GAS VALVE OPTION 2  HAS TO BE IMPLEMENTED ACCORDING TO CUSTOMIZED NEEDS in V4.07!
(not global released in V4.07, until sufficient pilot plant installation and testing, according email Hirzinger- Unterrainer, 28.05.2019)

ToDo:
-----

*******************************************************************************)
PROGRAM _CYCLIC

	(*--------------------------------------------------------------*)
	(* RESET of alarms and warnings and pre-settings				*)
	(*--------------------------------------------------------------*)
	bAMM_GT_AirSupply_Lo		:= FALSE;
	bAMM_GT_AirSupply_LoLo		:= FALSE;

	bAMM_DPr_GR_Baro_HiHi		:= FALSE;	(* A2261 *)

	bAMM_Pr_PCGT_Out_MS			:= FALSE;	(* W3448 *)

	bAMM_Pr_MGT_a_Filt_MS		:= FALSE;	(* W2462 *)
	bAMM_Pr_MGT_a_Filt_Lo		:= FALSE;	(* W2535 *)
	bAMM_Pr_MGT_a_Filt_LoLo		:= FALSE;	(* A2243 *)
	bAMM_Pr_MGT_a_Filt_Hi		:= FALSE;	(* W2536 *)
	bAMM_Pr_MGT_a_Filt_HiHi		:= FALSE;	(* A2246 *)
	bAMM_DPr_MGT_SetAct_Hi		:= FALSE;	(* W3444 *)
	bAMM_DPr_MGT_SetAct_HiHi	:= FALSE;	(* A3376 *)

	bAMM_Pr_PCGT_a_Filt_MS		:= FALSE;	(* W2465 *)
	bAMM_Pr_PCGT_a_Filt_Lo		:= FALSE;	(* W2537 *)	(*nicht verwendet*)
	bAMM_Pr_PCGT_a_Filt_LoLo	:= FALSE;	(* A2250 *)	(*nicht verwendet*)
	bAMM_Pr_PCGT_a_Filt_Hi		:= FALSE;	(* W2538 *)
	bAMM_Pr_PCGT_a_Filt_HiHi	:= FALSE;	(* A2251 *)
	bAMM_DPr_PCGT_SetAct_Hi		:= FALSE;	(* W3445 *)
	bAMM_DPr_PCGT_SetAct_HiHi	:= FALSE;	(* A3377 *)

	(* Reset set-/actual-pressure deviation calculation *)
	rDPr_MGT_SetAct				:= 0;
	rDPr_PCGT_SetAct			:= 0;

	(* Mapping of previous parameter for compatibility of visu *)
	Para.bPr_MGT_a_Filt_Exist	:= Para.bPr_GT1_Active;
	Para.rPr_MGT_a_Filt_Hi		:= Para.rPr_GT1_LimHi2;
	Para.rPr_MGT_a_Filt_HiHi	:= Para.rPr_GT1_LimHi1;
	Para.rPr_MGT_a_Filt_Lo		:= Para.rPr_GT1_LimLo2;
	Para.rPr_MGT_a_Filt_LoLo	:= Para.rPr_GT1_LimLo1;

	Para.bPr_PCGT_a_Filt_Exist  := Para.bPr_PCGT_Active;
	Para.rPr_PCGT_a_Filt_Hi		:= Para.rPr_PCGT_LimHi2;
	Para.rPr_PCGT_a_Filt_HiHi	:= Para.rPr_PCGT_LimHi1;
	Para.rPr_PCGT_a_Filt_Lo		:= Para.rPr_PCGT_LimLo2;
	Para.rPr_PCGT_a_Filt_LoLo	:= Para.rPr_PCGT_LimLo1;

	(*--------------------------------------------------------------*)
	(* gas valve			 		 								*)
	(*--------------------------------------------------------------*)
	xTON_GASV_08s(IN:= OUT_GT.tGV1_Open.Do,	PT:= T#8s);
	xTON_GASV_20s(IN:= OUT_GT.tGV1_Open.Do, PT:= T#20s);

	bGASV_Open_8s	:= xTON_GASV_08s.Q;											(* valve opened for  8 seconds *)
	bGASV_Open_20s	:= xTON_GASV_20s.Q;											(* valve opened for 20 seconds *)

	(*--------------------------------------------------------------*)
	(* Filterung charge pressure			 		 								*)
	(*--------------------------------------------------------------*)
	xFILTER_R_P2s_200ms(In := IN_GT.rPr_Ch_P2s_Avg_UF, Filter := 20);
	xFILTER_R_P2s_50ms(In := IN_GT.rPr_Ch_P2s_Avg_UF, Filter := 5);
	xFILTER_R_P2s_500ms(In := IN_GT.rPr_Ch_P2s_Avg_UF, Filter := 50);
	xFILTER_R_P2s_160ms(In := IN_GT.rPr_Ch_P2s_Avg_UF, Filter := 16);

	(*--------------------------------------------------------------*)
	(* Filtering H2 content			 		 								*)
	(*--------------------------------------------------------------*)
	IF Para.bGT_H2Active THEN
		bMSF_H2 := (NOT IN_GT.tGT_H2.GoodQual AND IN_GT.tPB2MM.bParaSetupOk AND NOT IN_GT.bH2_Bus_Active) OR
				   (NOT IN_GT.bH2_Bus_MSF AND IN_GT.tPB2MM.bParaSetupOk AND IN_GT.bH2_Bus_Active);
		(* Measurement signal failure H2 content self-retain *)
		bS_MSF_H2 := bMSF_H2 OR (bS_MSF_H2 AND NOT IN_GT.tAB2GT.bResetWarning);
	ELSE
		bMSF_H2 				:= FALSE;
		bS_MSF_H2				:= FALSE;
	END_IF;

	IF Para.tiFilterConst_H2 = 0 THEN
		xLCRPT1_H2.t := 0.001; (* Filter time constant [s] *)
	ELSE
		xLCRPT1_H2.t := TIME_TO_REAL(Para.tiFilterConst_H2) /1000; (* Filter time constant [s] *)
	END_IF;
	IF NOT Para.bGT_H2Active THEN	(* Switch to zero H2 value in case H2 content measurement is not active *)
		xLCRPT1_H2.x := 0;
	ELSIF bS_MSF_H2 THEN			(* Switch to default H2 value in case of measurement signal failure H2 content *)
		xLCRPT1_H2.x := Para.rGT_H2_DefVal;
	ELSIF NOT IN_GT.bH2_Bus_Active THEN
		xLCRPT1_H2.x := LIMIT(0, IN_GT.tGT_H2.Unfilt, 1);
	ELSE
		xLCRPT1_H2.x := LIMIT(0, IN_GT.rH2_Bus, 1);
	END_IF;
	xLCRPT1_H2();

	(************************************************************************************************************************************)
	(************************              				  error monitoring		 	             	           **************************)
	(************************************************************************************************************************************)
	IF IN_GT.tPB2MM.bParaSetupOk THEN

		(*----------------------------------------------------------*)
		(* measurement signal failure 								*)
		(*----------------------------------------------------------*)
		bAMM_Pr_MGT_a_Filt_MS		:= Para.bPr_MGT_a_Filt_Exist 	AND NOT IN_GT.tPr_MGT_a_Filt.GoodQual;						(* W2462 *)
		bAMM_Pr_PCGT_a_Filt_MS		:= Para.bPr_PCGT_a_Filt_Exist	AND NOT IN_GT.tPr_PCGT_a_Filt.GoodQual;						(* W2465 *)
		bAMM_Pr_PCGT_Out_MS			:= Para.bPr_PCGT_Out_Exist 		AND NOT IN_GT.tPr_PCGT_Out.GoodQual;						(* W3448 *)

		(* Release monitoring *)
		xTOF_AMM_Pr_MGT_a_Filt_MS(IN := bAMM_Pr_MGT_a_Filt_MS, 	PT:= T#10s);	(* TOF because of filtered signals *)
		xTOF_AMM_Pr_PCGT_a_Filt_MS(IN:= bAMM_Pr_PCGT_a_Filt_MS, PT:= T#10s);
		xTOF_AMM_Pr_PCGT_Out_MS(IN 	 := bAMM_Pr_PCGT_Out_MS, 	PT:= T#10s);

		bRelMon_Pr_MGT_a_Filt	:= Para.bPr_MGT_a_Filt_Exist   	AND NOT xTOF_AMM_Pr_MGT_a_Filt_MS.Q;
		bRelMon_Pr_PCGT_a_Filt	:= Para.bPr_PCGT_a_Filt_Exist   AND NOT xTOF_AMM_Pr_PCGT_a_Filt_MS.Q;
		bRelMon_Pr_PCGT_Out		:= Para.bPr_PCGT_Out_Exist   	AND NOT xTOF_AMM_Pr_PCGT_Out_MS.Q;

		(* Block engine start after 5 times W2462 *) (* SWAT Rel.2 *)
		xCTD_Start(CD:= IN_GT.bEng_Start_TC2, LOAD:= NOT MM2VIS.bMsg2462, PV:= 5);
		xSR_Block(SET1:= xCTD_Start.Q AND EDGENEG(IN_GT.tEng_Run.Do), RESET:= NOT MM2VIS.bMsg2462);
		OUT_GT.bAMM_Pr_MGT_a_Filt_BlockStart := xSR_Block.Q1;

		(* Block engine start after 5 times W2465 *) (* SWAT Rel.3 *)
		xCTD_Start2465(CD:= IN_GT.bEng_Start_TC2, LOAD:= NOT MM2VIS.bMsg2465, PV:= 5);
		xSR_Block2465(SET1:= xCTD_Start2465.Q AND EDGENEG(IN_GT.tEng_Run.Do), RESET:= NOT MM2VIS.bMsg2465);
		OUT_GT.bAMM_Pr_PCGT_a_Filt_BlockStart := xSR_Block2465.Q1;

		(*----------------------------------------------------------*)
		(* deviation gas rail pressure from barometric pressure MAX	*)
		(*----------------------------------------------------------*)
		xTON_FGDRPS(IN:= IN_GT.tPB2MM.bParaSetupOk, PT:= T#60s); 	(* because of barometric ramp up *)

		IF bN_EngAct_IsZero AND NOT IN_GT.tEng_Run.Do AND xTON_FGDRPS.Q THEN
			bAMM_DPr_GR_Baro_HiHi	:= rPr_GR_Avg > (IN_GT.rPr_Baro_Internal + 0.100) AND bRelMon_Pr_GR_Avg;(* 100 mbar *)		(* A2261 *)
		END_IF

		(*----------------------------------------------------------*)
		(* main gas train pressure after filter 					*)
		(*----------------------------------------------------------*)
		xGR_MINR_MGT_a_Filt(In	:= IN_GT.tPr_MGT_a_Filt.Ai, Gw:= Para.rPr_MGT_a_Filt_Lo, Hy:= 0.1);		(* hyst. = 100 mbar *)
		xGR_MAXR_MGT_a_Filt(In	:= IN_GT.tPr_MGT_a_Filt.Ai,	Gw:= Para.rPr_MGT_a_Filt_Hi, Hy:= 0.1);		(* hyst. = 100 mbar *)

		bAMM_Pr_MGT_a_Filt_Lo		:= xGR_MINR_MGT_a_Filt.Q 								AND bRelMon_Pr_MGT_a_Filt;			(* W2535 *)
		bAMM_Pr_MGT_a_Filt_Hi		:= xGR_MAXR_MGT_a_Filt.Q 								AND bRelMon_Pr_MGT_a_Filt;			(* W2536 *)
		bAMM_Pr_MGT_a_Filt_LoLo		:= (IN_GT.tPr_MGT_a_Filt.Ai < Para.rPr_MGT_a_Filt_LoLo)	AND bRelMon_Pr_MGT_a_Filt;			(* A2243 *)
		bAMM_Pr_MGT_a_Filt_HiHi		:= (IN_GT.tPr_MGT_a_Filt.Ai > Para.rPr_MGT_a_Filt_HiHi) AND bRelMon_Pr_MGT_a_Filt;			(* A2246 *)

		(*----------------------------------------------------------*)
		(* prechamber gas train pressure after filter 				*)
		(*----------------------------------------------------------*)
		xGR_MINR_PCGT_a_Filt(In	:= IN_GT.tPr_PCGT_a_Filt.Ai, Gw:= Para.rPr_PCGT_a_Filt_Lo, Hy:= 0.1);	(* hyst. = 100 mbar *)
		xGR_MAXR_PCGT_a_Filt(In	:= IN_GT.tPr_PCGT_a_Filt.Ai, Gw:= Para.rPr_PCGT_a_Filt_Hi, Hy:= 0.1);	(* hyst. = 100 mbar *)

		bAMM_Pr_PCGT_a_Filt_Lo		:= xGR_MINR_PCGT_a_Filt.Q 									AND bRelMon_Pr_PCGT_a_Filt;		(* W2537 *)
		bAMM_Pr_PCGT_a_Filt_Hi		:= xGR_MAXR_PCGT_a_Filt.Q 									AND bRelMon_Pr_PCGT_a_Filt;		(* W2538 *)
		bAMM_Pr_PCGT_a_Filt_LoLo	:= (IN_GT.tPr_PCGT_a_Filt.Ai < Para.rPr_PCGT_a_Filt_LoLo)	AND bRelMon_Pr_PCGT_a_Filt;		(* A2250 *)
		bAMM_Pr_PCGT_a_Filt_HiHi	:= (IN_GT.tPr_PCGT_a_Filt.Ai > Para.rPr_PCGT_a_Filt_HiHi)	AND bRelMon_Pr_PCGT_a_Filt;		(* A2251 *)

		(*----------------------------------------------------------*)
		(* gas train compressed air supply 							*)
		(*----------------------------------------------------------*)
		bAMM_GT_AirSupply_Lo		:= NOT IN_GT.tGT_AirSupply_LoLo.Di; 														(* W2570 - SWAT5 new *)															(* A2289 *)
	END_IF

	(************************************************************************************************************************************)
    (************************                                monitoring of load rejection                      **************************)
    (************************************************************************************************************************************)
    xTP_LoadReject(IN:= (p_ist_Old - (IN_GT.rP_Nom * IN_GT.rP_Act_Norm_Filt)) > 500.0, PT:= T#60s);

    (* Save actual power every second *)
    xTON_1000ms(IN:= NOT xTON_1000ms.Q, PT:= T#1000ms);

    IF xTON_1000ms.Q THEN p_ist_Old := (IN_GT.rP_Nom * IN_GT.rP_Act_Norm_Filt);	END_IF

	(************************************************************************************************************************************)
	(************************           					  main gas train  					 		       **************************)
	(************************************************************************************************************************************)

	(*--------------------------------------------------------------*)
	(* gas pressure SETPOINT calculation							*)
	(*--------------------------------------------------------------*)
	xRAMPE_R_DPr_MGT_P1(In		:= Para.rDPr_MGT_P1);			(* The parameters are delivered to the calculation via ramp *)
	xRAMPE_R_DPr_MGT_P2(In		:= Para.rDPr_MGT_P2);			(* ramp = 10 mbar/s *)
	xRAMPE_R_DPr_MGT_Ch_P1(In	:= Para.rDPr_MGT_Ch_P1);
	xRAMPE_R_DPr_MGT_Ch_P2(In	:= Para.rDPr_MGT_Ch_P2);

	IF NOT xEngType.Type9 THEN
		xSigScal_R_DPr_MGT_sp.X		:= IN_GT.rPr_Ch_P2s_Avg;
	ELSE
		xSigScal_R_DPr_MGT_sp.X		:= xFILTER_R_P2s_160ms.Out;
	END_IF

	xSigScal_R_DPr_MGT_sp.X1	:= xRAMPE_R_DPr_MGT_Ch_P1.Out;
	xSigScal_R_DPr_MGT_sp.X2	:= xRAMPE_R_DPr_MGT_Ch_P2.Out;
	xSigScal_R_DPr_MGT_sp.Y1	:= xRAMPE_R_DPr_MGT_P1.Out;
	xSigScal_R_DPr_MGT_sp.Y2	:= xRAMPE_R_DPr_MGT_P2.Out;
	xSigScal_R_DPr_MGT_sp();

	(* absolute --> relative *)
	IF xEngType.Type6 AND IN_GT.bGen2_Act AND IN_GT.tGCB_On.Di THEN
		rPr_MGT_sp				:= MIN(MAX(xFILTER_R_P2s_500ms.Out , IN_GT.rPr_Leanox_Set), (xFILTER_R_P2s_500ms.Out  + rPr_max_P2s_Offset)) + xSigScal_R_DPr_MGT_sp.Y_SCAL - IN_GT.rPr_Baro_Internal;
	ELSIF xEngType.Type9 AND IN_GT.bGen2_Act AND IN_GT.tGCB_On.Di THEN
		rPr_MGT_sp				:= MIN(MAX(xFILTER_R_P2s_160ms.Out , IN_GT.rPr_Leanox_Set), (xFILTER_R_P2s_160ms.Out  + rPr_max_P2s_Offset)) + xSigScal_R_DPr_MGT_sp.Y_SCAL - IN_GT.rPr_Baro_Internal;
	ELSE
		rPr_MGT_sp				:= xFILTER_R_P2s_500ms.Out + xSigScal_R_DPr_MGT_sp.Y_SCAL - IN_GT.rPr_Baro_Internal;
	END_IF;

	MM2VIS.rPr_MGT_sp			:= rPr_MGT_sp;	(* VISU *)

	(*--------------------------------------------------------------*)
	(* calculated gas pressure after main gas pressure regulator	*)
	(*--------------------------------------------------------------*)
	xSigScal_R_MGT_PipeLoss.X	:= IN_GT.rPr_Ch_P2s_Avg;
	xSigScal_R_MGT_PipeLoss.X1	:= Para.rPr_MGT_PipeLoss_Ch_P1;
	xSigScal_R_MGT_PipeLoss.X2	:= Para.rPr_MGT_PipeLoss_Ch_P2;
	xSigScal_R_MGT_PipeLoss.Y1	:= Para.rPr_MGT_PipeLoss_P1;
	xSigScal_R_MGT_PipeLoss.Y2	:= Para.rPr_MGT_PipeLoss_P2;
	xSigScal_R_MGT_PipeLoss();

	(* absolute --> relative *)
	IF OUT_GT.tGV1_Open.Do THEN
		rPr_MGT_Out_Calc		:= rPr_GR_Avg + xSigScal_R_MGT_PipeLoss.Y_SCAL - IN_GT.rPr_Baro_Internal;			(* VISU *)
	ELSE
		rPr_MGT_Out_Calc		:= 0;
	END_IF

	(*--------------------------------------------------------------*)
	(* set/actual gas pressure comparison							*)
	(*--------------------------------------------------------------*)
	(* calculation of set/actual gas pressure deviation *)
	IF OUT_GT.tGV1_Open.Do AND bRelMon_Pr_GR_Avg THEN
		rDPr_MGT_SetAct	:= rPr_MGT_Out_Calc - rPr_MGT_sp; 											(* VISU *)
	END_IF

	(* monitoring of set/actual gas pressure deviation *)
	IF bGASV_Open_20s AND NOT xTP_LoadReject.Q THEN
		bAMM_DPr_MGT_SetAct_Hi 		:= ABS(rDPr_MGT_SetAct) > 0.2 OR bMGT_SetActAdjust_Windup;		(* 200 mbar *)		(* W3444 *)
		bAMM_DPr_MGT_SetAct_HiHi	:= (ABS(rDPr_MGT_SetAct) > 0.4) AND NOT IN_GT.bPBC_Active; 		(* 400 mbar *)		(* A3376 *)		(* SWAT Rel. 5 *)
	END_IF

	IF IN_GT.tPB2MM.bParaSetupOk THEN
		bAMM_GT_AirSupply_LoLo		:= bAMM_DPr_MGT_SetAct_Hi AND NOT IN_GT.tGT_AirSupply_LoLo.Di;  (* A2289 *)
	END_IF;

	(*--------------------------------------------------------------*)
	(* set/actual gas pressure adjustment							*)
	(*--------------------------------------------------------------*)
	(* On-/off-switching of function only if engine isn't running *)
	IF bN_EngAct_IsZero THEN	bMGT_SetActAdjustActive_Save := Para.bMGT_SetActAdjustActive; END_IF

	IF IN_GT.tPB2MM.bParaSetupOk THEN	Para.bMGT_SetActAdjustActive := bMGT_SetActAdjustActive_Save; END_IF	(* parameter only changeable if engine isn't running *)

	IF Para.bMGT_SetActAdjustActive THEN

		(* time until next run of controller - Integralverstärkung *)
		xTON_MGT_SetActAdjust(IN:= bRel_MGT_SetActAdjust, PT:= T#1s);
		bRel_MGT_SetActAdjust	:= TRUE;

		(* duration of set/actual gas pressure adjustment *)
		xTP_MGT_SetActAdjust(IN	:= bGASV_Open_8s, 		  PT:= T#10s);

		IF 	xTP_MGT_SetActAdjust.Q 	AND	OUT_GT.tGV1_Open.Do AND
			xTON_MGT_SetActAdjust.Q			  				AND
			NOT bMGT_SetActAdjust_Windup 	  				AND
			bRelMon_Pr_GR_Avg
		THEN
			(* calculation of set/actual gas pressure deviation *)
			rDPr_MGT_SetAct_GR			:= (rPr_MGT_sp + IN_GT.rPr_Baro_Internal) - rPr_GR_Avg;

			(* Der maximal zulässige Ausgleichsauf- bzw. -abschlag beträgt 400mbar *)
			Perm.rDPr_MGT_SetActAdjust	:= LIMIT(-0.405, Perm.rDPr_MGT_SetActAdjust + (rDPr_MGT_SetAct_GR * 0.5), 0.405);
			bRel_MGT_SetActAdjust		:= FALSE;
		END_IF
	ELSE
		Perm.rDPr_MGT_SetActAdjust	:= 0;		(* RESET *)
	END_IF

	(*--------------------------------------------------------------*)
	(* FIXED gas pressure setpoint in case of emergency stop		*)
	(*--------------------------------------------------------------*)
	xTP_Pr_MGT_sp_fix(IN:= EDGENEG(OUT_GT.tGV1_Open.Do) AND (bGnlTrip1 OR bGnlTrip2), PT:= T#10s);

	IF xTP_Pr_MGT_sp_fix.Q	THEN 		(* fixed gas pressure of 130 mbar *)
		rPr_MGT_sp := 0.130;
		MM2VIS.rPr_MGT_sp := 0.130;
	ELSIF NOT OUT_GT.tGV1_Open.Do THEN 	(* engine is not running *)
		rPr_MGT_sp := 0;
		MM2VIS.rPr_MGT_sp := 0;
	ELSE 								(* controlled gas pressure setpoint *)
		rPr_MGT_sp := rPr_MGT_sp + Perm.rDPr_MGT_SetActAdjust;
	END_IF

	(*--------------------------------------------------------------*)
	(* handover gas pressure setpoint to AO		 					*)
	(*--------------------------------------------------------------*)
	OUT_GT.tPr_MGT_sp.Ao 		:=  rPr_MGT_sp - Para.rPr_MGT_sp_offset;
	bMGT_SetActAdjust_Windup	:= (OUT_GT.tPr_MGT_sp.Ao <= Para.rPr_MGT_spScalMin) OR (OUT_GT.tPr_MGT_sp.Ao >= Para.rPr_MGT_spScalMax);

	(************************************************************************************************************************************)
	(************************           			  main gas train - blow off valve			  		       **************************)
	(************************************************************************************************************************************)
	xTP_MGT_BOV_Open_Min(IN:= EDGENEG(OUT_GT.tGV1_Open.Do), PT:= Para.tiBOV_Open_Min);		(* mimimum opening time at shut down *)
	xTP_MGT_BOV_Open_Max(IN:= EDGENEG(OUT_GT.tGV1_Open.Do), PT:= Para.tiBOV_Open_Max);		(* maximum opening time at shut down *)

	(*--------------------------------------------------------------*)
	(* Deviation gas rail pressure from charging pressure			*)
	(*--------------------------------------------------------------*)
	IF IN_GT.bGT_GrC_Bloc THEN
		rDPr_GR_BOV_Open := 2.5;
	ELSE
		rDPr_GR_BOV_Open := Para.rDPr_GR_BOV_Open;
	END_IF;
	xGR_MAXR_DPr_GR_P2s(In:= rPr_GR_Avg - xFILTER_R_P2s_50ms.Out, Gw:= rDPr_GR_BOV_Open, Hy:= Para.rDPr_GR_BOV_Open_Hy);

	(* Gasrail is not allowed to be lower than the barometric pressure otherwise air could flow into the GasRail-> flammable mix *)
	IF (rPr_GR_Avg > IN_GT.rPr_Baro_Internal) THEN
		OUT_GT.tMGT_BOV.Do	:= 		xGR_MAXR_DPr_GR_P2s.Q  OR (* open on differential pressure between boost pressure and gas rail pressure *)
									(xTP_MGT_BOV_Open_Max.Q AND (* limit the opening duration to a maximum time *)
									(xTP_MGT_BOV_Open_Min.Q OR  (* limit the opening duration to a minimum time *)
									(rPr_GR_Avg > (IN_GT.rPr_Baro_Internal + 0.08)))); (* close on reaching barometric pressure plus offset *)
	ELSE
		OUT_GT.tMGT_BOV.Do	:= FALSE;
	END_IF

	(************************************************************************************************************************************)
	(************************            main gas train - pressure regulator dome blow off valve	            *************************)
	(************************************************************************************************************************************)

	(* Hysteresis for activating dome blow off valve on the gas rail set-act pressure deviation *)
	IF xEngType.Type6 THEN
		rDPr_MGT_DBOV_SetAct_GR_Hy := 0.25;
		rDPr_MGT_DBOV_SetAct_GR_Th := 0.30;
	ELSIF xEngType.Type9 THEN
		rDPr_MGT_DBOV_SetAct_GR_Hy := 0.05;
		rDPr_MGT_DBOV_SetAct_GR_Th := 0.50;
	ELSE
		rDPr_MGT_DBOV_SetAct_GR_Hy := 0.05;
		rDPr_MGT_DBOV_SetAct_GR_Th := 0.30;
	END_IF;

	xSR_DPr_MGT_DBOV_GR_SetAct.SET1 	:= rPr_MGT_Out_Calc - rPr_MGT_sp >= rDPr_MGT_DBOV_SetAct_GR_Th AND NOT IN_GT.bGT_GrC_Bloc;
	xSR_DPr_MGT_DBOV_GR_SetAct.RESET 	:= rPr_MGT_Out_Calc - rPr_MGT_sp < 	rDPr_MGT_DBOV_SetAct_GR_Th - rDPr_MGT_DBOV_SetAct_GR_Hy OR xTON_MGT_DBOV.Q OR IN_GT.bGT_GrC_Bloc;
	xSR_DPr_MGT_DBOV_GR_SetAct();
	xTON_MGT_DBOV(IN := xSR_DPr_MGT_DBOV_GR_SetAct.Q1);

	(* Activate dome blow off valve on positive edge of the main blow off valve for a certain time *)
	xSR_DBOV_MBOV_Logic_Ena(SET1 := EDGEPOS(xTP_LoadReject.Q), RESET := EDGENEG(xTP_LoadReject.Q) OR EDGENEG(OUT_GT.tMGT_BOV.Do));
	xTOF_POS_EDGE_MGT_BOV(IN := EDGEPOS(OUT_GT.tMGT_BOV.Do) AND xSR_DBOV_MBOV_Logic_Ena.Q1);

	(* Gasrail is not allowed to be lower than the barometric pressure otherwise air could flow into the GasRail-> flammable mix *)
	IF (rPr_GR_Avg > IN_GT.rPr_Baro_Internal) THEN
		OUT_GT.tMGT_DBOV.Do := 	(xSR_DPr_MGT_DBOV_GR_SetAct.Q1						(* open on set-act deviation of gas rail pressure *)
								OR xTOF_POS_EDGE_MGT_BOV.Q							(* open on positive edge of MBOV for a certain time *)
								OR IN_GT.bLR_Act_DBOV)								(* open on load rejection detection *)
								AND NOT IN_GT.bGT_GrC_Bloc;							(* disable during grid code event *)
	ELSE
		OUT_GT.tMGT_DBOV.Do	:= FALSE;
	END_IF

	(************************************************************************************************************************************)
	(************************           				  prechamber gas train  				 		       **************************)
	(************************************************************************************************************************************)

	(*--------------------------------------------------------------*)
	(* gas pressure SETPOINT calculation							*)
	(*--------------------------------------------------------------*)
	xRAMPE_R_DPr_PCGT_P1(In		:= Para.rDPr_PCGT_P1);			(* The parameters are delivered to the calculation via ramp *)
	xRAMPE_R_DPr_PCGT_P2(In		:= Para.rDPr_PCGT_P2);			(* ramp = 10 mbar/s *)
	xRAMPE_R_DPr_PCGT_Ch_P1(In	:= Para.rDPr_PCGT_Ch_P1);
	xRAMPE_R_DPr_PCGT_Ch_P2(In	:= Para.rDPr_PCGT_Ch_P2);

	xSigScal_R_DPr_PCGT_sp.X	:= IN_GT.rPr_Ch_P2s_Avg;
	xSigScal_R_DPr_PCGT_sp.X1	:= xRAMPE_R_DPr_PCGT_Ch_P1.Out;
	xSigScal_R_DPr_PCGT_sp.X2	:= xRAMPE_R_DPr_PCGT_Ch_P2.Out;
	xSigScal_R_DPr_PCGT_sp.Y1	:= xRAMPE_R_DPr_PCGT_P1.Out;
	xSigScal_R_DPr_PCGT_sp.Y2	:= xRAMPE_R_DPr_PCGT_P2.Out;
	xSigScal_R_DPr_PCGT_sp();

	(* absolute --> relative *)
	rPr_PCGT_sp					:= IN_GT.rPr_Ch_P2s_Avg + xSigScal_R_DPr_PCGT_sp.Y_SCAL - IN_GT.rPr_Baro_Internal;
	MM2VIS.rPr_PCGT_sp			:= IN_GT.rPr_Ch_P2s_Avg + xSigScal_R_DPr_PCGT_sp.Y_SCAL - IN_GT.rPr_Baro_Internal;	(* VISU *)

	(*--------------------------------------------------------------*)
	(* set/actual gas pressure comparison							*)
	(*--------------------------------------------------------------*)
	(* calculation of set/actual gas pressure deviation *)
	IF OUT_GT.tGV1_Open.Do AND bRelMon_Pr_PCGT_Out THEN
		rDPr_PCGT_SetAct		:= IN_GT.tPr_PCGT_Out.Ai - rPr_PCGT_sp; 											(* VISU *)
	END_IF

	(* monitoring of  set/actual gas pressure deviation *)
	xTON_bMsg3377_Active(IN:= (IN_GT.rP_Nom * IN_GT.rP_Act_Norm_Filt) > 2000, PT:= T#120s);		(* SWAT Rel.2 *)
	xSR_bMsg3377_Active(SET1:= IN_GT.bEng_Start_TC2, RESET:= xTON_bMsg3377_Active.Q);				(* SWAT Rel.2 *)
	IF bGASV_Open_20s AND NOT xTP_LoadReject.Q THEN
		xSigScal_R_SetAct_Hi.X		:= IN_GT.rPr_Ch_P2s_Avg;
		xSigScal_R_SetAct_Hi.X1		:= 0.5;			(*  500 mbar(abs) *)
		xSigScal_R_SetAct_Hi.X2		:= 7.0;			(* 7000 mbar(abs) *)
		xSigScal_R_SetAct_Hi.Y1		:= 0.2;			(*  200 mbar *)
		xSigScal_R_SetAct_Hi.Y2		:= 0.3;			(*  300 mbar *)
		xSigScal_R_SetAct_Hi();

		xSigScal_R_SetAct_HiHi.X	:= IN_GT.rPr_Ch_P2s_Avg;
		xSigScal_R_SetAct_HiHi.X1	:= 0.5;			(*  500 mbar(abs) *)
		xSigScal_R_SetAct_HiHi.X2	:= 7.0;			(* 7000 mbar(abs) *)
		xSigScal_R_SetAct_HiHi.Y1	:= 0.25;		(*  250 mbar *)
		xSigScal_R_SetAct_HiHi.Y2	:= 0.4;			(*  400 mbar *)
		xSigScal_R_SetAct_HiHi();

		bAMM_DPr_PCGT_SetAct_Hi 	:= ABS(rDPr_PCGT_SetAct) > xSigScal_R_SetAct_Hi.Y_SCAL OR bPCGT_SetActAdjust_Windup;		(* W3445 *)
		bAMM_DPr_PCGT_SetAct_HiHi	:= (ABS(rDPr_PCGT_SetAct) > xSigScal_R_SetAct_HiHi.Y_SCAL) AND xSR_bMsg3377_Active.Q1;		(* A3377 *)
	END_IF

	(* Delay time of W3445 *) (* SWAT Rel.5 *)
	xTON_DelayTrigger(IN:= IN_GT.tGCB_On.Di AND (IN_GT.rP_Act_Norm_Filt * IN_GT.rP_Nom) > 2000, PT:= T#120s);
	xSR_DelayTime(SET1:= xTON_DelayTrigger.Q, RESET:= IN_GT.bEng_Start);
	IF xSR_DelayTime.Q1 THEN
		tiDPr_PCGT_SetAct_Hi := T#250s;
	ELSE
		tiDPr_PCGT_SetAct_Hi := T#5s;
	END_IF

	(*--------------------------------------------------------------*)
	(* set/actual gas pressure adjustment							*)
	(*--------------------------------------------------------------*)
	(* On-/off-switching of function only if engine isn't running *)
	IF bN_EngAct_IsZero THEN	bPCGT_SetActAdjustActive_Save := Para.bPCGT_SetActAdjustActive;	END_IF

	IF IN_GT.tPB2MM.bParaSetupOk THEN	Para.bPCGT_SetActAdjustActive := bPCGT_SetActAdjustActive_Save; END_IF	(* parameter only changeable if engine isn't running *)

	IF Para.bPCGT_SetActAdjustActive THEN

		(* time until next run of controller - Integralverstärkung *)
		xTON_PCGT_SetActAdjust(IN:= bRel_PCGT_SetActAdjust, PT:= T#1s);
		bRel_PCGT_SetActAdjust	 := TRUE;

		(* duration of set/actual gas pressure adjustment *)
		xTP_PCGT_SetActAdjust(IN := bGASV_Open_8s, 			PT:= T#10s);

		IF 	xTP_PCGT_SetActAdjust.Q  AND OUT_GT.tGV1_Open.Do AND
			xTON_PCGT_SetActAdjust.Q 						 AND
			NOT bPCGT_SetActAdjust_Windup 					 AND
			bRelMon_Pr_PCGT_Out
		THEN
			(* calculation of set/actual gas pressure deviation *)
			rDPr_PCGT_SetAct_PCGT_Out	:= rPr_PCGT_sp - IN_GT.tPr_PCGT_Out.Ai;

			(* Der maximal zulässige Ausgleichsauf- bzw. -abschlag beträgt 400mbar *)
			Perm.rDPr_PCGT_SetActAdjust	:= LIMIT(-0.405, Perm.rDPr_PCGT_SetActAdjust + (rDPr_PCGT_SetAct_PCGT_Out * 0.5), 0.405);
			bRel_PCGT_SetActAdjust		:= FALSE;
		END_IF

	ELSE
		Perm.rDPr_PCGT_SetActAdjust	:= 0;		(* RESET *)
	END_IF

	(*--------------------------------------------------------------*)
	(* FIXED gas pressure setpoint in case of engine stop			*)
	(*--------------------------------------------------------------*)
	IF NOT OUT_GT.tGV1_Open.Do THEN		(* engine is not running *)
		rPr_PCGT_sp := 0;
		MM2VIS.rPr_PCGT_sp := 0;
	ELSE 								(* controlled gas pressure setpoint *)
		rPr_PCGT_sp := rPr_PCGT_sp + Perm.rDPr_PCGT_SetActAdjust;
	END_IF

	(*--------------------------------------------------------------*)
	(* handover gas pressure setpoint to AO		 					*)
	(*--------------------------------------------------------------*)
	OUT_GT.tPr_PCGT_sp.Ao 	  := rPr_PCGT_sp - Para.rPr_PCGT_sp_offset;
	bPCGT_SetActAdjust_Windup := (OUT_GT.tPr_PCGT_sp.Ao <= Para.rPr_PCGT_spScalMin) OR (OUT_GT.tPr_PCGT_sp.Ao >= Para.rPr_PCGT_spScalMax);

	(*--------------------------------------------------------------*)
	(* Option: gas valve position feedback		 					*) (* V4.07 *)
	(*--------------------------------------------------------------*)
	tGV_struct[1].alm_1sf := (	  OUT_GT.tGV1_Open.Do AND (NOT IN_GT.tGV1_Opened.Di AND IN_GT.tGV1_Opened.GoodQual) ) ;			(* Gas valve position detection opening failure (->error bit 1) *)
	tGV_struct[1].alm_0sf := (NOT OUT_GT.tGV1_Open.Do AND (NOT IN_GT.tGV1_Closed.Di AND IN_GT.tGV1_Closed.GoodQual) );			(* Gas valve position detection closing failure (->error bit 2)*)
	tGV_struct[1].alm_psf := ( (IN_GT.tGV1_Opened.Di AND IN_GT.tGV1_Opened.GoodQual) AND (IN_GT.tGV1_Closed.Di AND IN_GT.tGV1_Closed.GoodQual) );	(* Gas valve position detection failure (->error bit 3) *)
	tGV_struct[1].gv_status :=	BOOL_TO_DINT(tGV_struct[1].alm_1sf) *2 +			(* forward status for alarms and VIS: any value >1=failure message *)
								BOOL_TO_DINT(tGV_struct[1].alm_0sf) *4 +
								BOOL_TO_DINT(tGV_struct[1].alm_psf) *8 ;

	tGV_struct[2].alm_1sf := (	  OUT_GT.tGV2_Open.Do AND (NOT IN_GT.tGV2_Opened.Di AND IN_GT.tGV2_Opened.GoodQual) ) ;			(* Gas valve position detection opening failure (->error bit 1) *)
	tGV_struct[2].alm_0sf := (NOT OUT_GT.tGV2_Open.Do AND (NOT IN_GT.tGV2_Closed.Di AND IN_GT.tGV2_Closed.GoodQual) );			(* Gas valve position detection closing failure (->error bit 2) *)
	tGV_struct[2].alm_psf := ( (IN_GT.tGV2_Opened.Di AND IN_GT.tGV2_Opened.GoodQual) AND (IN_GT.tGV2_Closed.Di AND IN_GT.tGV2_Closed.GoodQual) );	(* Gas valve position detection failure (->error bit 3) *)
	tGV_struct[2].gv_status:=	BOOL_TO_DINT(tGV_struct[2].alm_1sf) *2 +			(* forward status for alarms and VIS: any value >1=failure message *)
								BOOL_TO_DINT(tGV_struct[2].alm_0sf) *4 +
								BOOL_TO_DINT(tGV_struct[2].alm_psf) *8 ;

	(* gv_Struct : 	STRUCT for local 'function like' processing in an array loop, without need for external .fun file    (*VERSION V4.07*)
	//enable : BOOL; (*from Parameter*)
	//on : BOOL; (*real position status*)
	//off : BOOL; (*real position status*)
	//man_off : BOOL; (*optional manual command*)
	//man_on : BOOL; (*optional manual command*)
	//command_on : BOOL; (*command to valve*)
	//command_off : BOOL; (*command to valve*)
	//...

	(*--------------------------------------------------------------------------*)
	(* Option: Upstream Customer Main Gas Valve control and position feedback	*) (*V4.09*)
	(*--------------------------------------------------------------------------*)
	OUT_GT.tGV_Upstream_Release.Do := (IN_GT.bEng_Aux_Dem_CDR 				(* Demanded Engine OR COOL DOWN RUN OR	*)
									OR IN_GT.tFastStartReq.Di )				(* V4.10 change issue #51  *)
								//	OR IN_GT.bReady4FastStart
								//	OR IN_GT.bReady4VeryFastStart) 			(* IF 562 OR IF563 Ready for fast start *)
								AND NOT IN_GT.bMsg1031			(* emergency stop *)
								AND NOT IN_GT.bMsg1052			(* gas prealarm  *)
								AND NOT IN_GT.bMsg1053			(* gas alarm *)
								AND NOT IN_GT.bMsg1054;			(* fire prealarm *)

	(* Para Option selective part for Upstream Customer Main Gas Valve *)
	IF Para.iGasTrain_Upstream_Type = 1 THEN		(* Para value '1' == Gas Valve Type with permanent release and feedback signals, e.g. Valpes/Bernard  (=option bit0) *)

		OUT_GT.tGV_Upstream_Open.Do := FALSE; //:= IN_GT.bEng_Aux_Dem_CDR   		(*  COOL DOWN RUN Verknüpfung 	Do open External Customer Gasvalve 	 *) (*OldName: NewPV *)

		tGV_struct[0].command_on	:= 	   OUT_GT.tGV_Upstream_Release.Do;  		(* FEHLT NOCH: COOL DOWN RUN Verknüpfung 	Do open External Customer Gasvalve 	 *) (*OldName: NewPV *)
	//	tGV_struct[0].command_off	:= NOT OUT_GT.tGV_Upstream_Open.Do;

		tGV_struct[0].on 	:=  IN_GT.tGV_Upstream_Opened.Di AND IN_GT.tGV_Upstream_Opened.GoodQual ;												(*	DI Gasvalve position status	 *) (*OldName: NewPV *)
		tGV_struct[0].off	:= (IN_GT.tGV_Upstream_Closed.Di AND IN_GT.tGV_Upstream_Closed.GoodQual)
						OR (NOT IN_GT.tGV_Upstream_Opened.Di AND IN_GT.tGV_Upstream_Opened.GoodQual AND NOT IN_GT.tGV_Upstream_Closed.GoodQual) ;	(*	DI Gasvalve position status	 *) (*OldName: NewPV *)

		tGV_struct[0].alm_1sf := (	  tGV_struct[0].command_on AND (NOT tGV_struct[0].on  AND IN_GT.tGV_Upstream_Opened.GoodQual) ); 	(* valve position detection opening failure(2) *)
		tGV_struct[0].alm_0sf := (NOT tGV_struct[0].command_on AND (NOT tGV_struct[0].off AND IN_GT.tGV_Upstream_Closed.GoodQual) ); 	(* valve position detection closing failure(4) *)
		tGV_struct[0].alm_psf := (    tGV_struct[0].on  AND tGV_struct[0].off  );														(* valve position detection failure (8) *)

	ELSIF Para.iGasTrain_Upstream_Type = 2 THEN 	(* Para value '2' == Gas Valve Type with permanent release +open pulse commands, e.g.Kromschroeter (=option bit1) *)
		xTON_MGV_Pos_Pulse(IN := OUT_GT.tGV_Upstream_Release.Do   		(*  Do Open External Customer Gasvalve continuous pulsing	 *)
									AND NOT IN_GT.tGV_Upstream_Opened.Di
									AND NOT xTON_MGV_Neg_Pulse.Q, PT := T#10s);
		xTON_MGV_Neg_Pulse(IN := xTON_MGV_Pos_Pulse.Q, PT :=  t#2s );
		OUT_GT.tGV_Upstream_Open.Do := xTON_MGV_Pos_Pulse.Q
								AND NOT IN_GT.bMsg1031			(* emergency stop *)
								AND NOT IN_GT.bMsg1052			(* gas prealarm  *)
								AND NOT IN_GT.bMsg1053			(* gas alarm *)
								AND NOT IN_GT.bMsg1054;			(* fire prealarm *)

		tGV_struct[0].command_on	:= 	   OUT_GT.tGV_Upstream_Release.Do;  		(* forward output state to display and supervise External Customer Gasvalve state	 *)
	//	tGV_struct[0].command_off	:= NOT OUT_GT.tGV_Upstream_Open.Do;

		tGV_struct[0].on 	:=  IN_GT.tGV_Upstream_Opened.Di AND IN_GT.tGV_Upstream_Opened.GoodQual ;								(*	DI Gasvalve position status	 *)
//		tGV_struct[0].off	:= (IN_GT.tGV_Upstream_Closed.Di AND IN_GT.tGV_Upstream_Closed.GoodQual)
//		OR (NOT IN_GT.tGV_Upstream_Opened.Di AND IN_GT.tGV_Upstream_Opened.GoodQual AND NOT IN_GT.tGV_Upstream_Closed.GoodQual)   ;	(*	DI Gasvalve position status	 *)

		tGV_struct[0].alm_1sf := (	  tGV_struct[0].command_on AND (NOT tGV_struct[0].on  AND IN_GT.tGV_Upstream_Opened.GoodQual) ); 	(* valve position detection opening failure (2) *)
//		tGV_struct[0].alm_0sf := (NOT tGV_struct[0].command_on AND (NOT tGV_struct[0].off AND IN_GT.tGV_Upstream_Closed.GoodQual) ); 	(* valve position detection closing failure (4) *)
//		tGV_struct[0].alm_psf := (    tGV_struct[0].on  AND tGV_struct[0].off  );  														(* valve position detection failure (8) *)

	ELSIF Para.iGasTrain_Upstream_Type = 4 THEN		(* parameter value = '4' == Customized Gas Valve Type ? for further use -  CURRENTLY UNDEFINED  (=option bit2)*)
		(* ToDo: Enter code variants for additional gasvalve designs here in future ! *)

	ELSE	(*V4.07.1 alternative path, if NO option bit selected (from Para.iGasTrain_Upstream_Type = '0') *)
		OUT_GT.tGV_Upstream_Release.Do	:= FALSE;
		OUT_GT.tGV_Upstream_Open.Do 	:= FALSE;
		tGV_struct[0].command_on		:= FALSE;
		tGV_struct[0].on 				:= FALSE ;
		tGV_struct[0].off				:= FALSE ;
		tGV_struct[0].alm_1sf 			:= FALSE ;
		tGV_struct[0].alm_0sf			:= FALSE ;
		tGV_struct[0].alm_psf			:= FALSE ;
		tGV_struct[0].gv_status			:= 0;
	END_IF

	(*status summary for VIS messages*)
	tGV_struct[0].gv_status:=	BOOL_TO_DINT(tGV_struct[0].command_on) + 		(* forward status for alarms and VIS: 0=closed, 1=open *)
								BOOL_TO_DINT(tGV_struct[0].alm_1sf) *2 +		(* forward status for alarms and VIS: any other value >1=failure message *)
								BOOL_TO_DINT(tGV_struct[0].alm_0sf) *4 +
								BOOL_TO_DINT(tGV_struct[0].alm_psf) *8 ;

END_PROGRAM
```

#### gas_trainInit.st
```iecst
(*******************************************************************************
gas_train		gas train  					(INIT)

This code is confidential and proprietary to the INNIO Company.
It may not be used in any form, or reproduced in any manner,
without the express written permission of the INNIO Company.
Copyright, INNIO Company, 2019

Customized modifications: -
------------------------

History:
-------
V3.30.0	06.11.2014	Tinello		Update to NEW specification

Instructions for use:
--------------------

*******************************************************************************)
PROGRAM _INIT

	(* ramp settings *)
	xRAMPE_R_DPr_MGT_P1.enable		:= TRUE;
	xRAMPE_R_DPr_MGT_P1.Rise		:= 0.010;		(* 10 mbar/s *)
	xRAMPE_R_DPr_MGT_P1.Sink		:= 0.010;		(* 10 mbar/s *)
	xRAMPE_R_DPr_MGT_P1.TC_Time		:= TASK_TIME_100MS;

	xRAMPE_R_DPr_MGT_P2.enable		:= TRUE;
	xRAMPE_R_DPr_MGT_P2.Rise		:= 0.010;		(* 10 mbar/s *)
	xRAMPE_R_DPr_MGT_P2.Sink		:= 0.010;		(* 10 mbar/s *)
	xRAMPE_R_DPr_MGT_P2.TC_Time		:= TASK_TIME_100MS;

	xRAMPE_R_DPr_MGT_Ch_P1.enable	:= TRUE;
	xRAMPE_R_DPr_MGT_Ch_P1.Rise		:= 0.010;		(* 10 mbar/s *)
	xRAMPE_R_DPr_MGT_Ch_P1.Sink		:= 0.010;		(* 10 mbar/s *)
	xRAMPE_R_DPr_MGT_Ch_P1.TC_Time	:= TASK_TIME_100MS;

	xRAMPE_R_DPr_MGT_Ch_P2.enable	:= TRUE;
	xRAMPE_R_DPr_MGT_Ch_P2.Rise		:= 0.010;		(* 10 mbar/s *)
	xRAMPE_R_DPr_MGT_Ch_P2.Sink		:= 0.010;		(* 10 mbar/s *)
	xRAMPE_R_DPr_MGT_Ch_P2.TC_Time	:= TASK_TIME_100MS;

	xRAMPE_R_DPr_PCGT_P1.enable		:= TRUE;
	xRAMPE_R_DPr_PCGT_P1.Rise		:= 0.010;		(* 10 mbar/s *)
	xRAMPE_R_DPr_PCGT_P1.Sink		:= 0.010;		(* 10 mbar/s *)
	xRAMPE_R_DPr_PCGT_P1.TC_Time	:= TASK_TIME_100MS;

	xRAMPE_R_DPr_PCGT_P2.enable		:= TRUE;
	xRAMPE_R_DPr_PCGT_P2.Rise		:= 0.010;		(* 10 mbar/s *)
	xRAMPE_R_DPr_PCGT_P2.Sink		:= 0.010;		(* 10 mbar/s *)
	xRAMPE_R_DPr_PCGT_P2.TC_Time	:= TASK_TIME_100MS;

	xRAMPE_R_DPr_PCGT_Ch_P1.enable	:= TRUE;
	xRAMPE_R_DPr_PCGT_Ch_P1.Rise	:= 0.010;		(* 10 mbar/s *)
	xRAMPE_R_DPr_PCGT_Ch_P1.Sink	:= 0.010;		(* 10 mbar/s *)
	xRAMPE_R_DPr_PCGT_Ch_P1.TC_Time	:= TASK_TIME_100MS;

	xRAMPE_R_DPr_PCGT_Ch_P2.enable	:= TRUE;
	xRAMPE_R_DPr_PCGT_Ch_P2.Rise	:= 0.010;		(* 10 mbar/s *)
	xRAMPE_R_DPr_PCGT_Ch_P2.Sink	:= 0.010;		(* 10 mbar/s *)
	xRAMPE_R_DPr_PCGT_Ch_P2.TC_Time	:= TASK_TIME_100MS;

	(* Settings for DBOV *)
	rDPr_MGT_DBOV_SetAct_GR_Th; 				(* gas rail pressure threshold for main gas train dome blow off valve *)
	rDPr_MGT_DBOV_SetAct_GR_Hy; 				(* gas rail pressure hysteresis for main gas train dome blow off valve different for type 6/9*)
	xTOF_POS_EDGE_MGT_BOV.PT		:= T#300ms; (* duration for opening DBOV after positive edge of MBOV *)
	xTON_MGT_DBOV.PT				:= T#60s;

	(* PT1 settings for H2 content measurement *)
	xLCRPT1_H2.enable := TRUE;
	xLCRPT1_H2.t	  := 1;

END_PROGRAM
```

#### gas_train.var
```iecst
VAR
	bGASV_Open_8s : BOOL := FALSE; (*Main gasvalve is opened for 8s*)
	bGASV_Open_20s : BOOL := FALSE; (*Main gasvalve is opened for 20s*)
	bMGT_SetActAdjustActive_Save : BOOL := FALSE; (*SAVE - main gas train set-/actual-pressure adjustment active*)
	bMGT_SetActAdjust_Windup : BOOL := FALSE; (*main gas train set-/actual-pressure adjustment controller - windup protection*)
	bPCGT_SetActAdjustActive_Save : BOOL := FALSE; (*SAVE - prechamber gas train set-/actual-pressure adjustment active*)
	bPCGT_SetActAdjust_Windup : BOOL := FALSE; (*prechamber gas train set-/actual-pressure adjustment controller - windup protection*)
	bRelMon_Pr_MGT_a_Filt : BOOL := FALSE; (*Release monitoring main gas train pressure after filter *)
	bRelMon_Pr_PCGT_a_Filt : BOOL := FALSE; (*Release monitoring prechamber gas train pressure after filter *)
	bRelMon_Pr_PCGT_Out : BOOL := FALSE; (*Release monitoring gas pressure after pre chamber gas pressure regulator*)
	bRel_MGT_SetActAdjust : BOOL := FALSE; (*release of set/actual gas pressure adjustment*)
	bRel_PCGT_SetActAdjust : BOOL := FALSE; (*release of set/actual gas pressure adjustment*)
	p_ist_Old : REAL := 0.0; (*SAVE actual power*)
	rDPr_MGT_SetAct_GR : REAL := 0.0; (*main gas train set-/actual-pressure deviation from gas rail [bar]*)
	rDPr_PCGT_SetAct_PCGT_Out : REAL := 0.0; (*main gas train set-/actual-pressure deviation from pressure after pre chamber gas pressure regulator [bar]*)
	rDPr_MGT_DBOV_SetAct_GR_Hy : REAL := 0.0; (* main gas train set-/actual-pressure deviation from gas rail hysteresis for dome blow off valve [bar] *)
	rDPr_MGT_DBOV_SetAct_GR_Th : REAL := 0.0; (* main gas train set-/actual-pressure deviation from gas rail threshold to activate dome blow off valve [bar] *)
END_VAR
VAR CONSTANT
	TASK_TIME_100MS : UINT := 100; (*Taskklassen Zeit 100ms *)
END_VAR
VAR
	xGR_MAXR_DPr_GR_P2s : GR_MAXR := (0); (*FuB*)
	xGR_MAXR_MGT_a_Filt : GR_MAXR := (0); (*FuB*)
	xGR_MAXR_PCGT_a_Filt : GR_MAXR := (0); (*FuB*)
	xGR_MINR_MGT_a_Filt : GR_MINR := (0); (*FuB*)
	xGR_MINR_PCGT_a_Filt : GR_MINR := (0); (*FuB*)
	xRAMPE_R_DPr_MGT_Ch_P1 : RAMPE_R := (0); (*FuB*)
	xRAMPE_R_DPr_MGT_Ch_P2 : RAMPE_R := (0); (*FuB*)
	xRAMPE_R_DPr_MGT_P1 : RAMPE_R := (0); (*FuB*)
	xRAMPE_R_DPr_MGT_P2 : RAMPE_R := (0); (*FuB*)
	xRAMPE_R_DPr_PCGT_Ch_P1 : RAMPE_R := (0); (*FuB*)
	xRAMPE_R_DPr_PCGT_Ch_P2 : RAMPE_R := (0); (*FuB*)
	xRAMPE_R_DPr_PCGT_P1 : RAMPE_R := (0); (*FuB*)
	xRAMPE_R_DPr_PCGT_P2 : RAMPE_R := (0); (*FuB*)
	xSigScal_R_DPr_PCGT_sp : xSigScal_R := (0); (*FuB - prechamber gas train - difference pressure setpoint [bar]*)
	xSigScal_R_MGT_PipeLoss : xSigScal_R := (0); (*FuB - main gas train - pressure loss of pipe [bar]*)
	xSigScal_R_SetAct_Hi : xSigScal_R := (0); (*FuB*)
	xSigScal_R_SetAct_HiHi : xSigScal_R := (0); (*FuB*)
	xTOF_AMM_Pr_MGT_a_Filt_MS : TOF := (0); (*FuB*)
	xTOF_AMM_Pr_PCGT_a_Filt_MS : TOF := (0); (*FuB*)
	xTOF_AMM_Pr_PCGT_Out_MS : TOF := (0); (*FuB*)
	xTON_1000ms : TON := (0); (*FuB*)
	xTON_FGDRPS : TON := (0); (*FuB*)
	xTON_GASV_08s : TON := (0); (*FuB*)
	xTON_GASV_20s : TON := (0); (*FuB*)
	xTON_MGT_SetActAdjust : TON := (0); (*FuB*)
	xTON_PCGT_SetActAdjust : TON := (0); (*FuB*)
	xTP_LoadReject : TP := (0); (*FuB*)
	xTP_MGT_BOV_Open_Max : TP := (0); (*FuB*)
	xTP_MGT_BOV_Open_Min : TP := (0); (*FuB*)
	xTP_MGT_SetActAdjust : TP := (0); (*FuB*)
	xTP_PCGT_SetActAdjust : TP := (0); (*FuB*)
	xTP_Pr_MGT_sp_fix : TP := (0); (*FuB*)
	xSR_Block : SR := (0);
	xSR_bMsg3377_Active : SR := (0); (*FuB*)
	xTON_bMsg3377_Active : TON := (0); (*FuB*)
	xSR_Block2465 : SR := (0);
	xTON_DelayTrigger : TON;
	xSR_DelayTime : SR;
	xTON_MGV_Pos_Pulse : TON;
	xTON_MGV_Neg_Pulse : TON;
	xTOF_POS_EDGE_MGT_BOV : TOF; (* Pulse to open the DBOV at positve EDGE of MBOV *)
	rDPr_GR_BOV_Open : REAL; (*main chamber difference pressure maximum - open blowoff valve [bar]*)
	xSR_DBOV_MBOV_Logic_Ena : SR; (* Enable opening of DBOV on pos edge of MBOV only once *)
	rPr_max_P2s_Offset : REAL := 0.5; (* p2s offset  for J6-Gen2 rPr_MGT_sp calculation *)
	xSR_DPr_MGT_DBOV_GR_SetAct : SR; (* main gas train dome blow off valve depending on gas rail pressure set/act deviation*)
	xTON_MGT_DBOV : TON; (* close DBOV if pressure deviation is not below hysteresis after delay *)
END_VAR
```

### Program Logical/Gastrain/biogas (IEC) - Biogas
